// Robot Parameter                         
UserData.DelayTime                         := _parCfg.Rob.Parameter.DelayTime;
UserData.WaitForNrOfCmd                    := _parCfg.Rob.Parameter.WaitForNrOfCmd;
UserData.WaitAtBlendingZone                := _parCfg.Rob.Parameter.WaitAtBlendingZone;
UserData.AllowSecSeqWhileSubprogram        := _parCfg.Rob.Parameter.AllowSecSeqWhileSubprogram;
UserData.AllowDynamicBlending              := _parCfg.Rob.Parameter.AllowDynamicBlending;
UserData.SyncReaction                      := _parCfg.Rob.Parameter.SyncReaction;
UserData.SyncDelay                         := _parCfg.Rob.Parameter.SyncDelay;
UserData.MessageLevel                      := _parcfg.Rob.Parameter.MessageLevel;

// ReadRobotData
UserData.RCManufacturer                    := AxesGroup.State.RobotData.RCManufacturer; 
UserData.RCOrderID                         := AxesGroup.State.RobotData.RCOrderID; 
UserData.RCSerialNumber                    := AxesGroup.State.RobotData.RCSerialNumber;
UserData.RASerialNumber                    := AxesGroup.State.RobotData.RASerialNumber;
UserData.RCFirmwareVersion                 := AxesGroup.State.RobotData.RCFirmwareVersion;

UserData.RCInterpreterVersion.MajorVersion := STRING_TO_USINT(MID(AxesGroup.State.RobotData.RCInterpreterVersion, LEN := 1, POS := 1));
UserData.RCInterpreterVersion.MinorVersion := STRING_TO_USINT(MID(AxesGroup.State.RobotData.RCInterpreterVersion, LEN := 1, POS := 2));
UserData.RCInterpreterVersion.PatchVersion := STRING_TO_USINT(MID(AxesGroup.State.RobotData.RCInterpreterVersion, LEN := 1, POS := 3));

UserData.AxisJointUsed                     := AxesGroup.State.RobotData.AxisJointUsed;
UserData.AxisExternalUsed                  := AxesGroup.State.RobotData.AxisExternalUsed;
UserData.AxisJointUnit                     := AxesGroup.State.RobotData.AxisJointUnit;
UserData.AxisExternalUnit                  := AxesGroup.State.RobotData.AxisExternalUnit;
UserData.RCSupportedFunctions              := AxesGroup.State.RobotData.RCSupportedFunctions;
                                           
UserData.BrakeTestRequired                 := AxesGroup.State.ConfigurationData.BrakeTestRequired;
UserData.PathAccuracyMode                  := AxesGroup.State.ConfigurationData.PathAccuracyMode;
UserData.AvoidSingularity                  := AxesGroup.State.ConfigurationData.AvoidSingularity;
UserData.ConstantVelocitySupported         := AxesGroup.State.ConfigurationData.ConstantVelocitySupported;
UserData.StepModeExactStopActive           := AxesGroup.State.ConfigurationData.StepModeExactStopActive;
UserData.StepModeBlendingActive            := AxesGroup.State.ConfigurationData.StepModeBlendingActive;
UserData.AcceleratingSupported             := AxesGroup.State.ConfigurationData.AcceleratingSupported;
UserData.DeceleratingSupported             := AxesGroup.State.ConfigurationData.DecceleratingSupported;
                                           
UserData.Initialized                       := Initialized;
UserData.Synchronized                      := Synchronized;
                                           
// Cyclic data                             
UserData.RCSRCIVersion                     := AxesGroup.Cyclic.RobToPlc.SRCIVersion;
UserData.IsMoving                          := AxesGroup.Cyclic.RobToPlc.StatusRobotArm.IsMoving;
UserData.PrimarySequencePaused             := AxesGroup.Cyclic.RobToPlc.StatusRobotArm.PrimarySequencePaused;
UserData.InPrimaryPos                      := AxesGroup.Cyclic.RobToPlc.StatusRobotArm.InPrimaryPos;
UserData.SecondarySequenceActive           := AxesGroup.Cyclic.RobToPlc.StatusRobotArm.SecondarySequenceActive;
UserData.ErrorPending                      := AxesGroup.Cyclic.RobToPlc.StatusRobotArm.ErrorPending;
UserData.RestartInProgress                 := AxesGroup.Cyclic.RobToPlc.StatusRobotArm.RestartInProgress;
UserData.Enabled                           := AxesGroup.Cyclic.RobToPlc.StatusRobotArm.Enabled;
UserData.Idle                              := AxesGroup.Cyclic.RobToPlc.StatusRobotArm.RaSequenceState = RaSequenceState.IDLE;
UserData.Executing                         := AxesGroup.Cyclic.RobToPlc.StatusRobotArm.RaSequenceState = RaSequenceState.EXECUTING;
UserData.Interrupted                       := AxesGroup.Cyclic.RobToPlc.StatusRobotArm.RaSequenceState = RaSequenceState.INTERRUPTED;
UserData.IsBlending                        := AxesGroup.Cyclic.RobToPlc.StatusRobotArm.IsBlending;  
UserData.OperationMode                     := AxesGroup.Cyclic.RobToPlc.StatusRobotArm.OperationMode;
UserData.CollisionDetectionEnabled         := AxesGroup.Cyclic.RobToPlc.StatusRobotArm.CollisionDetectedEnabled;
UserData.CollisionDetected                 := AxesGroup.Cyclic.RobToPlc.StatusRobotArm.CollisionDetected;
UserData.RestartRequested                  := AxesGroup.Cyclic.RobToPlc.StatusRobotArm.RestartRequested;
UserData.Accelerating                      := AxesGroup.Cyclic.RobToPlc.StatusRobotArm.Accelerating;
UserData.Decelerating                      := AxesGroup.Cyclic.RobToPlc.StatusRobotArm.Decelerating;
UserData.ConstantVelocity                  := AxesGroup.Cyclic.RobToPlc.StatusRobotArm.ConstantVelocity;
UserData.ActualOverride                    := PERCENT_UINT_TO_REAL( Value := AxesGroup.Cyclic.RobToPlc.Override, IsOptional := FALSE);

// Cyclic optional data
UserData.CartesianPosition                 := AxesGroup.CyclicOptional.RobToPlc.CartesianPosition;
UserData.ExtCartesianPosition              := AxesGroup.CyclicOptional.RobToPlc.CartesianPositionExt;  
UserData.JointPosition                     := AxesGroup.CyclicOptional.RobToPlc.JointPosition;
UserData.ExtJointPosition                  := AxesGroup.CyclicOptional.RobToPlc.JointPositionExt;

// Synchronizing
UserData.ToolDataSynchronizing             := AxesGroup.State.Synchronizing.Tool;
UserData.FrameDataSynchronizing            := AxesGroup.State.Synchronizing.Frame;
UserData.LoadDataSynchronizing             := AxesGroup.State.Synchronizing.Load;
UserData.WorkAreaDataSynchronizing         := AxesGroup.State.Synchronizing.WorkAreas;
UserData.SWLimitsSynchronizing             := AxesGroup.State.Synchronizing.SwLimits;
UserData.DefaultDynamicsSynchronizing      := AxesGroup.State.Synchronizing.DefaultDynamics;
UserData.ReferenceDynamicsSynchronizing    := AxesGroup.State.Synchronizing.ReferenceDynamics;


UserData.ActivateTwoSequences              := _parCfg.Com.TwoSequences;
UserData.ReadingCartesianPosition          :=  AxesGroup.State.ReadingCartesianPosition;
UserData.ReadingExtCartesianPosition       :=  AxesGroup.State.ReadingCartesianPositionExt;
UserData.ReadingJointPosition              :=  AxesGroup.State.ReadingJointPosition;
UserData.ReadingExtJointPosition           :=  AxesGroup.State.ReadingJointPositionExt;

                
END_METHOD

METHOD PRIVATE OnCall
VAR_IN_OUT
   /// Robot assignment of function
  AxesGroup : AxesGroup;
END_VAR
                  // map numeric value to enum, so that the corresponding message text is directly shown by the tooltip
ErrorIdEnum   := ErrorId;
WarningIdEnum := WarningId;
InfoIdEnum    := InfoId;

Error := HasError;

// Check Payload and In/Out data size
IF (( ROBOT_IN_DATA_SIZE  < 64 ) OR
    ( ROBOT_OUT_DATA_SIZE < 64 ))
THEN
  SetError(ErrorID := RobotLibraryErrorIdEnum.ERR_INVALID_LIBRARY_PARA, Overwrite := TRUE );
  RETURN;
END_IF


// Check AxesGroupID valid
IF (( AxesGroupID < RobotLibraryConstants.AXES_GROUP_ID_MIN ) OR
    ( AxesGroupID > RobotLibraryConstants.AXES_GROUP_ID_MAX ))
THEN
  SetError( ErrorID := RobotLibraryErrorIdEnum.ERR_INVALID_AXES_GROUP_ID, Overwrite := TRUE );
  RETURN;
END_IF


// Reset flag for initialization / Synchronization
IF ( Initialized OR Synchronized) AND ( AxesGroup.Cyclic.RobToPlc.TelegramState <> TelegramState.INITIALIZED)
THEN
  // Reset initialized flag
  Initialized := FALSE;
  // Reset Synchronized flag
  Synchronized := FALSE;
  // Set error 
  SetError( ErrorID := RobotLibraryErrorIdEnum.ERR_INIT_LOST_UNKNOWN_0x80A2, Overwrite := TRUE );
END_IF


// Warning for ACR Registers running low
IF ( AxesGroup.Acyclic.ActiveCommandRegister.CurrentAcrUsagePercent > RobotLibraryParameter.ACR_USAGE_WARNING_LIMIT )
THEN
  SetWarning( WarningID := RobotLibraryWarningIdEnum.WARN_ACR_FREE_ENTRIES_LOW, Overwrite := TRUE);  
END_IF

// Check ToolData boundary
IF ( AxesGroup.SystemData.ToolDataMin  <> 0 )  
THEN
  SetWarning( WarningID := RobotLibraryWarningIdEnum.WARN_TOOL_DATA_ARRAY_NOT_START_AT_ZERO, Overwrite := FALSE );
END_IF

// Check FrameData boundary
IF ( AxesGroup.SystemData.FrameDataMin <> 0 ) AND ( NOT HasWarning )  
THEN
  SetWarning( WarningID := RobotLibraryWarningIdEnum.WARN_FRAME_DATA_ARRAY_NOT_START_AT_ZERO, Overwrite := FALSE );
END_IF

// Check WorkAreas boundary
IF ( AxesGroup.SystemData.WorkAreasMin <> 0 ) AND ( NOT HasWarning )  
THEN
  SetWarning( WarningID := RobotLibraryWarningIdEnum.WARN_FRAME_DATA_ARRAY_NOT_START_AT_ZERO, Overwrite := FALSE);
END_IF


// Check configuration parameter changed ? 
CheckParameterChanged(AxesGroup := AxesGroup);
                
END_METHOD

METHOD OnExecRun : DINT
VAR_IN_OUT
  /// Robot assignment of function
  AxesGroup         : AxesGroup;
END_VAR
                  // building rising and falling edges
_enable_R( CLK := Enable);
_enable_F( CLK := Enable);

IF ( _enable_F.Q)
THEN
  Reset(AxesGroup := AxesGroup);
END_IF


OnExecRun := RobotLibraryConstants.RUNNING;

CASE _stepCmd OF
  
  00:  IF ( _enable_R.Q )
       THEN
         // Create log entry
         CreateLogMessage ( Timestamp   := SystemTime,
                            MessageType := MessageType.CMD,
                            Severity    := Severity.INFO,
                            MessageCode := 0,
                            MessageText := 'Robot Task Enabled');
       
         // reset the rising edge
        _enable_R();
         // set busy flag
         Busy := TRUE;
         // set timeout
         SetTimeout(PT := _timeoutCmd, rTimer := _timerCmd);
         // Reset FastStop       
         AxesGroup.Cyclic.PlcToRob.FastStop := 0;
         // Reset Active command register
         AxesGroup.Acyclic.ActiveCommandRegister.Reset();
       
         // check parameter valid
         IF ( CheckParameterValid(AxesGroup := AxesGroup) )
         THEN
           // take configuration parameter if not yet enabled
          _parCfg := ParCfg;
           // inc step counter
          _stepCmd := _stepCmd + 1; 
         END_IF
       END_IF
     
  01:  CASE AxesGroup.Cyclic.RobToPlc.TelegramState  OF

         TelegramState.UNDEFINED : ;
         
         TelegramState.ERROR_161_TELEGRAM_CONTROL_MISMATCH_TELEGRAM_STATE..TelegramState.ERROR_172_TELEGRAM_NUMBER_NOT_SUPPORTED:

           // clear error
           AxesGroup.Cyclic.PlcToRob.Control := ControlHalfByte.ACK_ERROR;        
           AxesGroup.Cyclic.PlcToRob.Control := ControlHalfByte.RESET; // always a reset, so that on the robot side the ACR is reseted         

         TelegramState.ERROR_173_SERVER_CONNECTION_LOST:

           // Reset interface including the ACR register on server side
           AxesGroup.Cyclic.PlcToRob.Control := ControlHalfByte.RESET;        
           
         TelegramState.READY_TO_RESUME :  
         
           // Resume
           AxesGroup.Cyclic.PlcToRob.Control := ControlHalfByte.RESUME;        
         
         TelegramState.READY_FOR_INITIALIZATION: 

           // Request initialization
           AxesGroup.Cyclic.PlcToRob.Control := ControlHalfByte.INITIALIZE;
           
         TelegramState.INITIALIZED: 

           // Reset Telegram Control 
           AxesGroup.Cyclic.PlcToRob.Control := ControlHalfByte.NONE;
           
           // Check SRCI Version is compatible ? 
           IF ( AxesGroup.Cyclic.RobToPlc.SRCIVersion.MajorVersion = RobotLibraryConstants.SRCIVersion.MajorVersion )
           THEN
             // set timeout
             SetTimeout(PT := _timeoutCmd, rTimer := _timerCmd);
             // inc step counter
            _stepCmd := _stepCmd + 1; 
           ELSE
             // set error 
             ErrorID     := RobotLibraryErrorIdEnum.ERR_SRCI_MAJOR_VERSION_INCOMPATIBLE_0x80A4;
             ErrorAddTxt := CONCAT('_stepCmd = ' , DINT_TO_STRING(_stepCmd));
           END_IF

       ELSE
         // TelegrammState in error          
         SetError( ErrorID := RobotLibraryErrorIdEnum.ERR_INIT_LOST_UNKNOWN_0xA2, Overwrite := TRUE );
         ErrorAddTxt := CONCAT('_stepCmd = ' , DINT_TO_STRING(_stepCmd));
       END_CASE

       // timeout exceeded ? 
       IF (CheckTimeout(_timerCmd) = RobotLibraryConstants.OK)
       THEN
         // Check Telegram State error ? 
         IF (( AxesGroup.Cyclic.RobToPlc.TelegramState >= TelegramState.ERROR_161_TELEGRAM_CONTROL_MISMATCH_TELEGRAM_STATE ) OR
             ( AxesGroup.Cyclic.RobToPlc.TelegramState <= TelegramState.ERROR_173_SERVER_CONNECTION_LOST                   ))
         THEN
           ErrorID     := AxesGroup.Cyclic.RobToPlc.TelegramState;
           ErrorAddTxt := CONCAT('_stepCmd = ' , DINT_TO_STRING(_stepCmd));
         ELSE
           ErrorID     := RobotLibraryErrorIdEnum.ERR_TIMEOUT_CMD;
           ErrorAddTxt := CONCAT('_stepCmd = ' , DINT_TO_STRING(_stepCmd));
         END_IF
       END_IF

       
  02: IF (( NOT _readMessages.Busy  ) AND 
          ( NOT _readMessages.Error )) 
      THEN
        // start function block
       _readMessages.Enable := TRUE;
       _readMessages.ParCmd.MsgID := 0;
       _readMessages.ParCmd.MessageLevel := _parCfg.Rob.Parameter.MessageLevel;
        
        // set timeout
        SetTimeout(PT := _timeoutCmd, rTimer := _timerCmd);
        // inc step counter
       _stepCmd := _stepCmd + 1;       
      ELSE
        // check error ? 
        IF (_readMessages.Error)
        THEN
          ErrorID     := _readMessages.ErrorID;
          ErrorAddTxt := _readMessages.ErrorAddTxt;;
        END_IF  
        // timeout exceeded ? 
        IF (CheckTimeout(_timerCmd) = RobotLibraryConstants.OK)
        THEN
          ErrorID     := RobotLibraryErrorIdEnum.ERR_TIMEOUT_CMD;
          ErrorAddTxt := CONCAT('_stepCmd = ' , DINT_TO_STRING(_stepCmd));
        END_IF
      END_IF
  
  03: IF ((     _readMessages.Enabled ) AND
          ( NOT _readMessages.Error   ))
      THEN       
        // --------------------------------------------------------------- 
        // !!! ReadMessages must stay active for the Message mechanism !!!
        // --------------------------------------------------------------- 
        // ReadMessages.Enable := FALSE;  
        // set timeout
        SetTimeout(PT := _timeoutCmd, rTimer := _timerCmd);
        // inc step counter
       _stepCmd := _stepCmd + 1;
      ELSE
         // check error ? 
         IF (_readMessages.Error)
         THEN
           ErrorID     := _readMessages.ErrorID;
           ErrorAddTxt := _readMessages.ErrorAddTxt;;
         END_IF  
       
         // timeout exceeded ? 
         IF (CheckTimeout(_timerCmd) = RobotLibraryConstants.OK)
         THEN
           ErrorID     := RobotLibraryErrorIdEnum.ERR_TIMEOUT_CMD;
           ErrorAddTxt := CONCAT('_stepCmd = ' , DINT_TO_STRING(_stepCmd));
         END_IF
       END_IF       
       
       
  04: IF (( NOT _exchangeConfiguration.Busy  ) AND 
          ( NOT _exchangeConfiguration.Error ))
      THEN
        // set command parameter
       _exchangeConfiguration.ParCmd.LogLevel                           :=  LogLevel; 
       _exchangeConfiguration.ParCmd.WaitAtBlendingZone                 := _parCfg.Rob.Parameter.WaitAtBlendingZone;
       _exchangeConfiguration.ParCmd.AllowSecSeqWhileSubprogram         := _parCfg.Rob.Parameter.AllowSecSeqWhileSubprogram;
       _exchangeConfiguration.ParCmd.AllowDynamicBlending               := _parCfg.Rob.Parameter.AllowDynamicBlending;
       _exchangeConfiguration.ParCmd.DelayTime                          := _parCfg.Rob.Parameter.DelayTime;
       _exchangeConfiguration.ParCmd.WaitForNrOfCmd                     := _parCfg.Rob.Parameter.WaitForNrOfCmd;
       _exchangeConfiguration.ParCmd.LifeSignTimeOut                    :=  TIME_TO_UINT(_parCfg.Com.LifeSignTimeOut);
       _exchangeConfiguration.ParCmd.SyncDelay                          := _parCfg.Rob.Parameter.SyncDelay;
       _exchangeConfiguration.ParCmd.SyncReaction                       := _parCfg.Rob.Parameter.SyncReaction;
       _exchangeConfiguration.ParCmd.DataEnableSync                     :=  SyncModesToDataEnableSync(Value := _parCfg.Plc.Parameter.SynchronizationModes);
       _exchangeConfiguration.ParCmd.DataInSync.ToolsInSync             :=  FALSE;
       _exchangeConfiguration.ParCmd.DataInSync.FramesInSync            :=  FALSE;
       _exchangeConfiguration.ParCmd.DataInSync.LoadsInSync             :=  FALSE;
       _exchangeConfiguration.ParCmd.DataInSync.WorkAreasInSync         :=  FALSE;
       _exchangeConfiguration.ParCmd.DataInSync.SoftwareLimitsInSync    :=  FALSE;
       _exchangeConfiguration.ParCmd.DataInSync.DefaultDynamicsInSync   :=  FALSE;
       _exchangeConfiguration.ParCmd.DataInSync.ReferenceDynamicsInSync :=  FALSE;         
       
        // start function block
       _exchangeConfiguration.Enable := TRUE;
        // set timeout
        SetTimeout(PT := _timeoutCmd, rTimer := _timerCmd);
        // inc step counter
       _stepCmd := _stepCmd + 1;       
      ELSE
        // check error ? 
        IF (_exchangeConfiguration.Error)
        THEN
          ErrorID     := _exchangeConfiguration.ErrorID;
          ErrorAddTxt := _exchangeConfiguration.ErrorAddTxt;;
        END_IF  
       
        // timeout exceeded ? 
        IF (CheckTimeout(_timerCmd) = RobotLibraryConstants.OK)
        THEN
          ErrorID     := RobotLibraryErrorIdEnum.ERR_TIMEOUT_CMD;
          ErrorAddTxt := CONCAT('_stepCmd = ' , DINT_TO_STRING(_stepCmd));
        END_IF
      END_IF
  
  
  05: IF ((     _exchangeConfiguration.Enabled ) AND
          ( NOT _exchangeConfiguration.Error   ))
      THEN     
        // --------------------------------------------------------------------- 
        // !!! ExchangeConfiguration must stay active for the Sync mechanism !!!
        // --------------------------------------------------------------------- 
        // ExchangeConfiguration.Enable := FALSE;  
        // set timeout
        SetTimeout(PT := _timeoutCmd, rTimer := _timerCmd);
        // inc step counter
       _stepCmd := _stepCmd + 1;       
      ELSE
        // check error ? 
        IF (_exchangeConfiguration.Error)
        THEN
          ErrorID     := _exchangeConfiguration.ErrorID;
          ErrorAddTxt := _exchangeConfiguration.ErrorAddTxt;;
        END_IF  
       
        // timeout exceeded ? 
        IF (CheckTimeout(_timerCmd) = RobotLibraryConstants.OK)
        THEN
          ErrorID     := RobotLibraryErrorIdEnum.ERR_TIMEOUT_CMD;
          ErrorAddTxt := CONCAT('_stepCmd = ' , DINT_TO_STRING(_stepCmd));
        END_IF
      END_IF

       
  06: IF (( NOT _readRobotData.Busy  ) AND 
          ( NOT _readRobotData.Error )) 
      THEN
        // start function block
       _readRobotData.Execute := TRUE;
        // set timeout
        SetTimeout(PT := _timeoutCmd, rTimer := _timerCmd);
        // inc step counter
       _stepCmd := _stepCmd + 1;       
      ELSE
        // check error ? 
        IF (_readRobotData.Error)
        THEN
          ErrorID     := _readRobotData.ErrorID;
          ErrorAddTxt := _readRobotData.ErrorAddTxt;;
        END_IF  
        // timeout exceeded ? 
        IF (CheckTimeout(_timerCmd) = RobotLibraryConstants.OK)
        THEN
          ErrorID     := RobotLibraryErrorIdEnum.ERR_TIMEOUT_CMD;
          ErrorAddTxt := CONCAT('_stepCmd = ' , DINT_TO_STRING(_stepCmd));
        END_IF
      END_IF
    
  
  07: IF ((     _readRobotData.Done  ) AND
          ( NOT _readRobotData.Busy  ) AND
          ( NOT _readRobotData.Error ))          
      THEN       
        // set initialized flag
        Initialized := TRUE;       
        // start function block
       _readRobotData.Execute := FALSE;
        // set timeout
        SetTimeout(PT := _timeoutCmd, rTimer := _timerCmd);
        // inc step counter
       _stepCmd := _stepCmd + 1;
       ELSE
         // check error ? 
         IF (_readRobotData.Error)
         THEN
           ErrorID     := _readRobotData.ErrorID;
           ErrorAddTxt := _readRobotData.ErrorAddTxt;;
         END_IF  
       
         // timeout exceeded ? 
         IF (CheckTimeout(_timerCmd) = RobotLibraryConstants.OK)
         THEN
           ErrorID     := RobotLibraryErrorIdEnum.ERR_TIMEOUT_CMD;
           ErrorAddTxt := CONCAT('_stepCmd = ' , DINT_TO_STRING(_stepCmd));
         END_IF
       END_IF

       
  08:  // Update Initialized state
       Initialized := NOT ERROR AND NOT Synchronized; {warning 'ToDo'}
       Initialized := NOT Synchronized;

       // Wait for task disable
       IF ( NOT Enable)
       THEN
         // Reset active command register
         AxesGroup.Acyclic.ActiveCommandRegister.Reset();
         // reset internal variables
         Reset(AxesGroup := AxesGroup);
         // Reset step counter
        _stepCmd := 0;         
         // finished okay
         OnExecRun := RobotLibraryConstants.OK;
       END_IF  

       
ELSE
  // invalid step
  ErrorID     := RobotLibraryErrorIdEnum.ERR_INVALID_STEP;
  ErrorAddTxt := CONCAT('_stepCmd = ' , DINT_TO_STRING(_stepCmd));
END_CASE
                
END_METHOD

METHOD PRIVATE ParseRecvPayload
VAR_IN_OUT
  /// Robot assignment of function
  AxesGroup   : AxesGroup;
  /// Inputs of PLC for communication from RC
  RobotInData : ARRAY[*] OF BYTE;
END_VAR
                  // reset all variables and payload
RecvData.Reset();
// Call RecvData FB, update payload and size 
RecvData(Payload := RobotInData, PayloadSize := ROBOT_IN_DATA_SIZE);

// check new data to receive ? 
IF ( Telegram.RobToPlc.Sequence[0].Header.SEQ_ACK <> AxesGroup.State.LastACK[0]) {warning 'ToDo: handle 2nd sequence'} 
THEN
  // delete old telegram data 
  SysDepMemSet(pDest := ADR(Telegram.RobToPlc), Value := 0 , DataLen := SIZEOF(Telegram.RobToPlc));
END_IF


ParseRecvPayloadHeader        ( AxesGroup := AxesGroup);
ParseRecvPayloadCyclic        ( AxesGroup := AxesGroup);
ParseRecvPayloadCyclicOptional( AxesGroup := AxesGroup);
ParseRecvPayloadSequence      ( AxesGroup := AxesGroup);
ParseRecvPayloadFooter        ( AxesGroup := AxesGroup);
ParseRecvPayloadLogging       ( AxesGroup := AxesGroup);


AxesGroup.State.LastACK[0] := Telegram.RobToPlc.Sequence[0].Header.SEQ_ACK; 
AxesGroup.State.LastACK[1] := Telegram.RobToPlc.Sequence[1].Header.SEQ_ACK; 
                
END_METHOD

METHOD PRIVATE ParseRecvPayloadCyclic
VAR_IN_OUT
  /// Robot assignment of function
  AxesGroup: AxesGroup;
END_VAR
                  
                
END_METHOD

METHOD PRIVATE ParseRecvPayloadCyclicOptional
VAR_IN_OUT
  /// Robot assignment of function
  AxesGroup    : AxesGroup;
END_VAR

VAR 
  /// internal index for loops
 _idx : DINT;
END_VAR
                  // AxesGroup.OptionalCyclic.RobToPlc.SubProgramData {{{
IF ( AxesGroup.CyclicOptional.RobToPlc.SubProgramData.Active )
THEN
  FOR _idx := 0 TO 25 {warning 'Add contant for DataMax'}
  DO
    Telegram.RobToPlc.CyclicOptional.SubProgramData.Data[_idx] := RecvData.GetByte(); 
  END_FOR
END_IF
// }}}
  
// AxesGroup.OptionalCyclic.RobToPlc.CartesianPos {{{
IF ( AxesGroup.CyclicOptional.RobToPlc.CartesianPosition.Active )
THEN
  Telegram.RobToPlc.CyclicOptional.CartesianPosition.X                    := RecvData.GetReal();
  Telegram.RobToPlc.CyclicOptional.CartesianPosition.Y                    := RecvData.GetReal();
  Telegram.RobToPlc.CyclicOptional.CartesianPosition.Z                    := RecvData.GetReal();
  Telegram.RobToPlc.CyclicOptional.CartesianPosition.Rx                   := RecvData.GetReal();
  Telegram.RobToPlc.CyclicOptional.CartesianPosition.Ry                   := RecvData.GetReal();
  Telegram.RobToPlc.CyclicOptional.CartesianPosition.Rz                   := RecvData.GetReal();
  Telegram.RobToPlc.CyclicOptional.CartesianPosition.Config               := RecvData.GetWord();
  Telegram.RobToPlc.CyclicOptional.CartesianPosition.Turns_J2_J1          := RecvData.GetByte();
  Telegram.RobToPlc.CyclicOptional.CartesianPosition.Turns_J4_J3          := RecvData.GetByte();
  Telegram.RobToPlc.CyclicOptional.CartesianPosition.Turns_J6_J5          := RecvData.GetByte();
  Telegram.RobToPlc.CyclicOptional.CartesianPosition.Turns_E1             := RecvData.GetByte();  
  Telegram.RobToPlc.CyclicOptional.CartesianPosition.E1                   := RecvData.GetReal();  
  Telegram.RobToPlc.CyclicOptional.CartesianPosition.ToolNo               := RecvData.GetUsint();
  Telegram.RobToPlc.CyclicOptional.CartesianPosition.FrameNo              := RecvData.GetUsint();
  Telegram.RobToPlc.CyclicOptional.CartesianPosition.CurrentlyUsedToolNo  := RecvData.GetUsint();
  Telegram.RobToPlc.CyclicOptional.CartesianPosition.CurrentlyUsedFrameNo := RecvData.GetUsint();
  Telegram.RobToPlc.CyclicOptional.CartesianPosition.Reserve_1            := RecvData.GetByte();
  Telegram.RobToPlc.CyclicOptional.CartesianPosition.Reserve_2            := RecvData.GetByte();  
END_IF
// }}}

// AxesGroup.OptionalCyclic.RobToPlc.JointPosition {{{
IF ( AxesGroup.CyclicOptional.RobToPlc.JointPosition.Active )
THEN
  Telegram.RobToPlc.CyclicOptional.JointPosition.J1         := RecvData.GetReal();
  Telegram.RobToPlc.CyclicOptional.JointPosition.J2         := RecvData.GetReal();
  Telegram.RobToPlc.CyclicOptional.JointPosition.J3         := RecvData.GetReal();
  Telegram.RobToPlc.CyclicOptional.JointPosition.J4         := RecvData.GetReal();
  Telegram.RobToPlc.CyclicOptional.JointPosition.J5         := RecvData.GetReal();
  Telegram.RobToPlc.CyclicOptional.JointPosition.J6         := RecvData.GetReal();
  Telegram.RobToPlc.CyclicOptional.JointPosition.E1         := RecvData.GetReal();
  Telegram.RobToPlc.CyclicOptional.JointPosition.E1_Reserve := RecvData.GetWord();
END_IF  
// }}}

// AxesGroup.OptionalCyclic.RobToPlc.CartesianForce {{{
IF ( AxesGroup.CyclicOptional.RobToPlc.Force.Active )
THEN
  Telegram.RobToPlc.CyclicOptional.Force.X  := RecvData.GetReal();
  Telegram.RobToPlc.CyclicOptional.Force.Y  := RecvData.GetReal();
  Telegram.RobToPlc.CyclicOptional.Force.Z  := RecvData.GetReal();
  Telegram.RobToPlc.CyclicOptional.Force.Rx := RecvData.GetReal();
  Telegram.RobToPlc.CyclicOptional.Force.Ry := RecvData.GetReal();
  Telegram.RobToPlc.CyclicOptional.Force.Rz := RecvData.GetReal();
END_IF  
// }}}    
  
// AxesGroup.OptionalCyclic.RobToPlc.Current {{{
IF ( AxesGroup.CyclicOptional.RobToPlc.Current.Active )
THEN
  Telegram.RobToPlc.CyclicOptional.Current.J1  := RecvData.GetReal();
  Telegram.RobToPlc.CyclicOptional.Current.J2  := RecvData.GetReal();
  Telegram.RobToPlc.CyclicOptional.Current.J3  := RecvData.GetReal();
  Telegram.RobToPlc.CyclicOptional.Current.J4  := RecvData.GetReal();
  Telegram.RobToPlc.CyclicOptional.Current.J5  := RecvData.GetReal();
  Telegram.RobToPlc.CyclicOptional.Current.J6  := RecvData.GetReal();
END_IF    
  
// AxesGroup.OptionalCyclic.RobToPlc.CartesianPosExt {{{
IF ( AxesGroup.CyclicOptional.RobToPlc.CartesianPositionExt.Active )
THEN
  Telegram.RobToPlc.CyclicOptional.CartesianPositionExt.E2 := RecvData.GetReal();
  Telegram.RobToPlc.CyclicOptional.CartesianPositionExt.E3 := RecvData.GetReal();
  Telegram.RobToPlc.CyclicOptional.CartesianPositionExt.E4 := RecvData.GetReal();
  Telegram.RobToPlc.CyclicOptional.CartesianPositionExt.E5 := RecvData.GetReal();
  Telegram.RobToPlc.CyclicOptional.CartesianPositionExt.E6 := RecvData.GetReal();
END_IF  
// }}}       
  
// AxesGroup.OptionalCyclic.RobToPlc.JointPosition {{{
IF ( AxesGroup.CyclicOptional.RobToPlc.JointPositionExt.Active )
THEN
  Telegram.RobToPlc.CyclicOptional.JointPositionExt.E2 := RecvData.GetReal();
  Telegram.RobToPlc.CyclicOptional.JointPositionExt.E3 := RecvData.GetReal();
  Telegram.RobToPlc.CyclicOptional.JointPositionExt.E4 := RecvData.GetReal();
  Telegram.RobToPlc.CyclicOptional.JointPositionExt.E5 := RecvData.GetReal();
  Telegram.RobToPlc.CyclicOptional.JointPositionExt.E6 := RecvData.GetReal();  
END_IF  
// }}}    
      
// AxesGroup.OptionalCyclic.RobToPlc.CartesianForceExt {{{
IF ( AxesGroup.CyclicOptional.RobToPlc.ForceExt.Active )
THEN
  Telegram.RobToPlc.CyclicOptional.ForceExt.E1  := RecvData.GetReal();
  Telegram.RobToPlc.CyclicOptional.ForceExt.E2  := RecvData.GetReal();
  Telegram.RobToPlc.CyclicOptional.ForceExt.E3  := RecvData.GetReal();
  Telegram.RobToPlc.CyclicOptional.ForceExt.E4  := RecvData.GetReal();
  Telegram.RobToPlc.CyclicOptional.ForceExt.E5  := RecvData.GetReal();
  Telegram.RobToPlc.CyclicOptional.ForceExt.E6  := RecvData.GetReal();
END_IF
// }}}    
  
// AxesGroup.OptionalCyclic.RobToPlc.CurrentExt {{{
IF ( AxesGroup.CyclicOptional.RobToPlc.CurrentExt.Active )
THEN
  Telegram.RobToPlc.CyclicOptional.CurrentExt.E1  := RecvData.GetReal();
  Telegram.RobToPlc.CyclicOptional.CurrentExt.E2  := RecvData.GetReal();
  Telegram.RobToPlc.CyclicOptional.CurrentExt.E3  := RecvData.GetReal();
  Telegram.RobToPlc.CyclicOptional.CurrentExt.E4  := RecvData.GetReal();
  Telegram.RobToPlc.CyclicOptional.CurrentExt.E5  := RecvData.GetReal();
  Telegram.RobToPlc.CyclicOptional.CurrentExt.E6  := RecvData.GetReal();
END_IF
// }}}
                
END_METHOD

METHOD PRIVATE ParseRecvPayloadFooter
VAR_IN_OUT
  /// Robot assignment of function
  AxesGroup : AxesGroup;
END_VAR
                  Telegram.RobToPlc.Footer.LifeSign := RecvData.GetLifeSignFooter(); 

                
END_METHOD

METHOD PRIVATE ParseRecvPayloadHeader
VAR_IN_OUT
  /// Robot assignment of function
  AxesGroup    : AxesGroup;
END_VAR
                  // Version
Telegram.RobToPlc.Header.SRCIVersion := ByteToVersion(RecvData.GetByte());
// Connection alive signal
Telegram.RobToPlc.Header.LifeSign    := RecvData.GetHalfeByte2(IncPayloadPtr := TRUE);
// Reserved byte
Telegram.RobToPlc.Header.Reserved       := RecvData.GetByte();
// Initialization and Telegram control state
Telegram.RobToPlc.Header.TelegramState  := RecvData.GetUsint();
// Combination of various RA related states.
Telegram.RobToPlc.Header.StatusRobotArm := RecvData.GetDword();
// Actual override in percentage encoding 
Telegram.RobToPlc.Header.Override       := RecvData.GetUint();
                
END_METHOD

METHOD PRIVATE ParseRecvPayloadLogging
VAR_IN_OUT
  /// Robot assignment of function
  AxesGroup    : AxesGroup;
END_VAR

VAR
  /// internal sequence index for loops
  _seqIdx : DINT;
  /// internal fragment index for loops
  _fragIdx : DINT;
END_VAR
                  RETURN;
FOR _seqIdx := 0 TO AxesGroup.State.SequenceCountRecv
DO
  // check new data to receive ? 
  IF ( Telegram.RobToPlc.Sequence[_seqIdx].Header.SEQ_ACK <> AxesGroup.State.LastACK[_seqIdx]) 
  THEN
    // Check sequence payload > 0 ?    
    IF (Telegram.RobToPlc.Sequence[_seqIdx].Header.PayloadLength > 0)
    THEN
      // Create log entry
      CreateLogMessagePara4 ( Timestamp   := SystemTime,
                              MessageType := MessageType.CMD,
                              Severity    := Severity.DEBUG,
                              MessageCode := 0,
                              MessageText := 'RecvData: ACK = {1}, received Sequence [{2}] with PayloadLength = {3}, Lifesign = {4}',
                              Para1       :=  UINT_TO_STRING(Telegram.RobToPlc.Sequence[_seqIdx].Header.SEQ_ACK),
                              Para2       :=  DINT_TO_STRING(_seqIdx),
                              Para3       :=  UINT_TO_STRING(Telegram.RobToPlc.Sequence[_seqIdx].Header.PayloadLength),
                              Para4       :=  BYTE_TO_STRING(Telegram.RobToPlc.Header.LifeSign));
  
      FOR _fragIdx := 0 TO AxesGroup.State.FragmentCountRecv[_seqIdx] 
      DO
        // Check fragment payload > 0 ?    
        IF (Telegram.RobToPlc.Sequence[_seqIdx].Fragment[_fragIdx].Header.PayloadLength > 0)
        THEN
          // Create log entry
          CreateLogMessagePara5 ( Timestamp   := SystemTime,
                                  MessageType := MessageType.CMD,
                                  Severity    := Severity.DEBUG,
                                  MessageCode := 0,
                                  MessageText := 'RecvData: received Fragment [{1}] with PayloadLength = {2}, CmdID <{3}> , CmdState: {4}, Fragment-Action Bits: {5}',
                                  Para1       :=  DINT_TO_STRING(0), {warning 'Add seqIdx'}
                                  Para2       :=  UINT_TO_STRING              (Telegram.RobToPlc.Sequence[_seqIdx].Fragment[_fragIdx].Header.PayloadLength),
                                  Para3       :=  DINT_TO_STRING              (Telegram.RobToPlc.Sequence[_seqIdx].Fragment[_fragIdx].Header.CmdID),
                                  Para4       :=  CMD_MESSAGE_STATE_TO_STRING (Telegram.RobToPlc.Sequence[_seqIdx].Fragment[_fragIdx].Command.Header.State),
                                  Para5       :=    FRAGMENT_ACTION_TO_STRING (Telegram.RobToPlc.Sequence[_seqIdx].Fragment[_fragIdx].Header.FragmentAction));
        END_IF
      END_FOR    
    END_IF
  END_IF
END_FOR  
                
END_METHOD

METHOD PRIVATE ParseRecvPayloadSequence
VAR_IN_OUT
  /// Robot assignment of function
  AxesGroup        : AxesGroup;
END_VAR

VAR
  /// internal index
 _idx              : DINT;
  /// index for sequence
 _seqIdx           : DINT;
  /// index for fragment
 _fragIdx          : DINT; 
  /// current payload pointer for current fragment
 _payLoadPtr       : DINT;
  /// Amount of sequences
 _seqCount         : DINT;
  /// current payload pointer of the current sequence
 _seqPayloadPtr    : UINT; 
END_VAR
                  // Check 2nd sequence active ? 
IF ( _parCfg.Com.TwoSequences )
THEN
 _seqCount := _seqCount + 1;
END_IF

FOR _seqIdx := 0 TO _seqCount
DO
  // Check 2nd sequence ? -> goto 2nd sequence payload address  
  IF ( _seqIdx = SECONDARY_SEQUENCE )
  THEN
    RecvData.PayloadPtr := CalculateSequencePayloadStartAdr(AxesGroup := AxesGroup, 
                                                            Direction := ComDirection.ROB_TO_PLC,
                                                            Sequence  := SequenceFlag.SECONDARY_SEQUENCE);
	END_IF

  // parste sequence header
  Telegram.RobToPlc.Sequence[_seqIdx].Header.SEQ_ACK       := RecvData.GetUint();
  Telegram.RobToPlc.Sequence[_seqIdx].Header.PayloadLength := RecvData.GetUint();
  
  // check new data available ? 
  IF ( Telegram.RobToPlc.Sequence[_seqIdx].Header.SEQ_ACK <> AxesGroup.State.LastACK[_seqIdx]) 
  THEN
    // Check sequence payload available ? 
    IF (Telegram.RobToPlc.Sequence[_seqIdx].Header.PayloadLength > 0)
    THEN
      // Check sequence payload length is valid ? 
      IF ( Telegram.RobToPlc.Sequence[_seqIdx].Header.PayloadLength > _parCfg.Com.TelegramLengthRobToPlc )
      THEN 
        // Create log entry for payload not valid 
        CreateLogMessagePara2 ( Timestamp   := SystemTime,
                                MessageType := MessageType.CMD,
                                Severity    := Severity.DEBUG,
                                MessageCode := 0,
                                MessageText := 'Invalid sequence payload length, Sequence = {1}, PayloadLength = {2} ',
                                Para1       :=  DINT_TO_STRING(_seqIdx),
                                Para2       :=  UINT_TO_STRING(Telegram.RobToPlc.Sequence[_seqIdx].Header.PayloadLength));
                                RETURN;
      ELSE
        // Create log entry
        CreateLogMessagePara4 ( Timestamp   := SystemTime,
                                MessageType := MessageType.CMD,
                                Severity    := Severity.DEBUG,
                                MessageCode := 0,
                                MessageText := 'RecvData: ACK = {1}, received Sequence [{2}] with PayloadLength = {3}, Lifesign = {4}',
                                Para1       :=  UINT_TO_STRING(Telegram.RobToPlc.Sequence[_seqIdx].Header.SEQ_ACK),
                                Para2       :=  DINT_TO_STRING(_seqIdx),
                                Para3       :=  UINT_TO_STRING(Telegram.RobToPlc.Sequence[_seqIdx].Header.PayloadLength),
                                Para4       :=  BYTE_TO_STRING(Telegram.RobToPlc.Header.LifeSign));
      END_IF
    
      // processing sequence payload                                  
      WHILE ( _seqPayloadPtr < Telegram.RobToPlc.Sequence[_seqIdx].Header.PayloadLength )
      DO                        
        // parse header
        Telegram.RobToPlc.Sequence[_seqIdx].Fragment[_fragIdx].Header.CmdID          := RecvData.GetUint();
        Telegram.RobToPlc.Sequence[_seqIdx].Fragment[_fragIdx].Header.Reserve        := RecvData.GetByte();
        Telegram.RobToPlc.Sequence[_seqIdx].Fragment[_fragIdx].Header.FragmentAction := RecvData.GetByte();
        Telegram.RobToPlc.Sequence[_seqIdx].Fragment[_fragIdx].Header.PayloadPointer := RecvData.GetUint();
        Telegram.RobToPlc.Sequence[_seqIdx].Fragment[_fragIdx].Header.PayloadLength  := RecvData.GetUint();
       
        // add header size to payload pointer 
       _seqPayloadPtr := _seqPayloadPtr + SIZEOF(Telegram.RobToPlc.Sequence[_seqIdx].Fragment[_fragIdx].Header);
        
        // Check fragment payload available ? 
        IF (Telegram.RobToPlc.Sequence[_seqIdx].Fragment[_fragIdx].Header.PayloadLength > 0)
        THEN
          // Check fragment payload length is valid ? 
          IF ( Telegram.RobToPlc.Sequence[_seqIdx].Fragment[_fragIdx].Header.PayloadLength > _parCfg.Com.TelegramLengthRobToPlc )
          THEN 
            // Create log entry for payload not valid 
            CreateLogMessagePara2 ( Timestamp   := SystemTime,
                                    MessageType := MessageType.CMD,
                                    Severity    := Severity.DEBUG,
                                    MessageCode := 0,
                                    MessageText := 'Invalid fragment payload length, Sequence = {1}, PayloadLength = {2} ',
                                    Para1       :=  DINT_TO_STRING(_seqIdx),
                                    Para2       :=  UINT_TO_STRING(Telegram.RobToPlc.Sequence[_seqIdx].Fragment[_fragIdx].Header.PayloadLength));
                                    RETURN;
          END_IF
        
          // Fill Response payload
          FOR _idx := 0 TO Telegram.RobToPlc.Sequence[_seqIdx].Fragment[_fragIdx].Header.PayloadLength -1
          DO
            // calculate payload pointer
           _payLoadPtr := Telegram.RobToPlc.Sequence[_seqIdx].Fragment[_fragIdx].Header.PayloadPointer + _idx;
          
            IF (( _payLoadPtr >= 0                                          ) AND
                ( _payLoadPtr <= RobotLibraryParameter.RESPONSE_PAYLOAD_MAX ))
            THEN  
              Telegram.RobToPlc.Sequence[_seqIdx].Fragment[_fragIdx].Command.Payload[_payLoadPtr] := RecvData.GetByte();
              // inc payload pointer
             _seqPayloadPtr := _seqPayloadPtr + SIZEOF(BYTE);
            ELSE
              // Create log entry for payload pointer not valid 
              CreateLogMessagePara3 ( Timestamp   := SystemTime,
                                      MessageType := MessageType.CMD,
                                      Severity    := Severity.DEBUG,
                                      MessageCode := 0,
                                      MessageText := 'Invalid fragment payload pointer, Sequence = {1}, Fragment = {2}, PayloadPointer = {3} ',
                                      Para1       :=  DINT_TO_STRING(_seqIdx),
                                      Para2       :=  DINT_TO_STRING(_fragIdx),
                                      Para3       :=  DINT_TO_STRING(_payLoadPtr));
                                      RETURN;
					  END_IF
           
          END_FOR
          
          // Add Response to ACR
          AxesGroup.Acyclic.ActiveCommandRegister.AddRsp(Telegram.RobToPlc.Sequence[_seqIdx].Fragment[_fragIdx]);
        
          // Only for debugging - header is part of the payload itself
          Telegram.RobToPlc.Sequence[_seqIdx].Fragment[_fragIdx].Command.Header.State                 :=      GetHalfeByteLo( Value :=  Telegram.RobToPlc.Sequence[_seqIdx].Fragment[_fragIdx].Command.Payload[0]);
          Telegram.RobToPlc.Sequence[_seqIdx].Fragment[_fragIdx].Command.Header.ParSeq                :=      GetHalfeByteHi( Value :=  Telegram.RobToPlc.Sequence[_seqIdx].Fragment[_fragIdx].Command.Payload[0]);
          Telegram.RobToPlc.Sequence[_seqIdx].Fragment[_fragIdx].Command.Header.AlarmMessageSeverity  :=        BYTE_TO_SINT(           Telegram.RobToPlc.Sequence[_seqIdx].Fragment[_fragIdx].Command.Payload[1]);
          Telegram.RobToPlc.Sequence[_seqIdx].Fragment[_fragIdx].Command.Header.AlarmMessageCode      :=  CombineBytesToUint( HiByte := Telegram.RobToPlc.Sequence[_seqIdx].Fragment[_fragIdx].Command.Payload[2],
                                                                                                                              LoByte := Telegram.RobToPlc.Sequence[_seqIdx].Fragment[_fragIdx].Command.Payload[3]);
          // Create log entry
          CreateLogMessagePara5 ( Timestamp   := SystemTime,
                                  MessageType := MessageType.CMD,
                                  Severity    := Severity.DEBUG,
                                  MessageCode := 0,
                                  MessageText := 'RecvData: received Fragment [{1}] with PayloadLength = {2}, CmdID <{3}> , CmdState: {4}, Fragment-Action Bits: {5}',
                                  Para1       :=  DINT_TO_STRING(_seqIdx),
                                  Para2       :=  UINT_TO_STRING              (Telegram.RobToPlc.Sequence[_seqIdx].Fragment[_fragIdx].Header.PayloadLength),
                                  Para3       :=  DINT_TO_STRING              (Telegram.RobToPlc.Sequence[_seqIdx].Fragment[_fragIdx].Header.CmdID),
                                  Para4       :=  CMD_MESSAGE_STATE_TO_STRING (Telegram.RobToPlc.Sequence[_seqIdx].Fragment[_fragIdx].Command.Header.State),
                                  Para5       :=    FRAGMENT_ACTION_TO_STRING (Telegram.RobToPlc.Sequence[_seqIdx].Fragment[_fragIdx].Header.FragmentAction));
        END_IF
        
        // Check still payload left ? -> goto next fragment  
        IF ( _seqPayloadPtr < Telegram.RobToPlc.Sequence[_seqIdx].Header.PayloadLength )
        THEN
         _fragIdx := _fragIdx + 1;        
        END_IF
        
        // Check fragment index limit reached ? 
        IF ( _fragIdx > RobotLibraryParameter.FRAGMENT_MAX ) 
        THEN 
          // Create log entry
          CreateLogMessagePara1 ( Timestamp   := SystemTime,
                                  MessageType := MessageType.CMD,
                                  Severity    := Severity.DEBUG,
                                  MessageCode := 0,
                                  MessageText := 'Fragment index out of range, _fragIdx = {1} ',
                                  Para1       :=  DINT_TO_STRING(_fragIdx));
                                  RETURN;
        END_IF        
      END_WHILE    
    END_IF
  END_IF    
END_FOR  
                
END_METHOD

METHOD Reset
VAR_IN_OUT
  /// Robot assignment of function
  AxesGroup : AxesGroup;  
END_VAR
                  // reset flags
Busy              := FALSE;
Initialized       := FALSE;
Synchronized      := FALSE;
Error             := FALSE;
ErrorID           := 0;
ErrorAddTxt       := '';
WarningID         := 0;
InfoID            := 0;  

// Reset internal functon blocks
_exchangeConfiguration      .Enable  := FALSE;
_readRobotData              .Execute := FALSE;
_readMessages               .Enable  := FALSE;  
_readToolData               .Execute := FALSE;  
_readFrameData              .Execute := FALSE;  
_readLoadData               .Execute := FALSE;  
_readWorkArea               .Execute := FALSE;  
_readRobotSWLimits          .Execute := FALSE;  
_readRobotDefaultDynamics   .Execute := FALSE;  
_readRobotReferenceDynamics .Execute := FALSE;  
_writeToolData              .Execute := FALSE;   
_writeFrameData             .Execute := FALSE;   
_writeLoadData              .Execute := FALSE;   
_writeWorkArea              .Execute := FALSE;   
_writeRobotSWLimits         .Execute := FALSE;   
_writeRobotDefaultDynamics  .Execute := FALSE;   
_writeRobotReferenceDynamics.Execute := FALSE;   

// Set Client error to force server error
AxesGroup.Cyclic.PlcToRob.Control := ControlHalfByte.NONE;

// Reset synchronisation state variables
AxesGroup.State.SyncStatePlc.InSync.Frame             := FALSE;
AxesGroup.State.SyncStatePlc.InSync.Tool              := FALSE;
AxesGroup.State.SyncStatePlc.InSync.Load              := FALSE;
AxesGroup.State.SyncStatePlc.InSync.WorkArea          := FALSE;
AxesGroup.State.SyncStatePlc.InSync.SwLimits          := FALSE;
AxesGroup.State.SyncStatePlc.InSync.DefaultDynamics   := FALSE;
AxesGroup.State.SyncStatePlc.InSync.ReferenceDynamics := FALSE;

AxesGroup.State.SyncStatePlc.UnSyncNo.Frame    := 0;
AxesGroup.State.SyncStatePlc.UnSyncNo.Tool     := 0;
AxesGroup.State.SyncStatePlc.UnSyncNo.Load     := 0;
AxesGroup.State.SyncStatePlc.UnSyncNo.WorkArea := 0;

AxesGroup.State.SyncStateRc .InSync.Frame             := FALSE;
AxesGroup.State.SyncStateRc .InSync.Tool              := FALSE;
AxesGroup.State.SyncStateRc .InSync.Load              := FALSE;
AxesGroup.State.SyncStateRc .InSync.WorkArea          := FALSE;
AxesGroup.State.SyncStateRc .InSync.SwLimits          := FALSE;
AxesGroup.State.SyncStateRc .InSync.DefaultDynamics   := FALSE;
AxesGroup.State.SyncStateRc .InSync.ReferenceDynamics := FALSE;

AxesGroup.State.SyncStateRc .UnSyncNo.Frame    := 0;
AxesGroup.State.SyncStateRc .UnSyncNo.Tool     := 0;
AxesGroup.State.SyncStateRc .UnSyncNo.Load     := 0;
AxesGroup.State.SyncStateRc .UnSyncNo.WorkArea := 0;

// Reset active command register
AxesGroup.Acyclic.ActiveCommandRegister.Reset();
      
// reset step counters
_stepCmd                   := 0;
_stepSyncFrameData         := 0;
_stepSyncLoadData          := 0;
_stepSyncDefaultDynamics   := 0;
_stepSyncReferenceDynamics := 0;
_stepSyncSWLimits          := 0;
_stepSyncToolData          := 0;
_stepSyncWorkArea          := 0;
                
END_METHOD

METHOD PUBLIC SetError
VAR_INPUT
  /// ErrorID reported by RC for error identification according to Table 7-1
  ErrorID   : WORD;
  /// TRUE = overwrite an existing error 
  Overwrite : BOOL;
END_VAR
                  IF ( NOT HasError ) OR ( Overwrite )
THEN
  THIS^.ErrorID := ErrorID;
END_IF
                
END_METHOD

METHOD PUBLIC SetInfo
VAR_INPUT
  /// InfoID for info identification reported during execution of command according to Table 7-5
  InfoID    : WORD;
  /// TRUE = overwrite an existing info 
  Overwrite : BOOL;
END_VAR
                  IF ( NOT HasInfo ) OR ( Overwrite )
THEN
  THIS^.InfoID := InfoID;
END_IF
                
END_METHOD

METHOD PUBLIC SetWarning
VAR_INPUT
  /// WarningID for warning identification reported during execution of command according to Table 7-3
  WarningID : WORD;
  /// TRUE = overwrite an existing warning 
  Overwrite : BOOL;
END_VAR
                  IF ( NOT HasWarning ) OR ( Overwrite )
THEN
  THIS^.WarningID := WarningID;
END_IF
                
END_METHOD

PROPERTY PROTECTED HasError : Bool
GET
VAR
END_VAR
                    HasError := ErrorID <> RobotLibraryErrorIdEnum.NO_ERROR;
                  
END_GET
END_PROPERTY

PROPERTY PROTECTED HasInfo : BOOL
GET
VAR
END_VAR
                    HasInfo := InfoID <> RobotLibraryInfoIdEnum.NO_INFO;
                  
END_GET
END_PROPERTY

PROPERTY PROTECTED HasWarning : BOOL
GET
VAR
END_VAR
                    HasWarning := WarningID <> RobotLibraryWarningIdEnum.NO_WARNING;
                  
END_GET
END_PROPERTY
END_FUNCTION_BLOCK

/// Switch operation mode of RC (Automatic External, T1 External, T2 External)
FUNCTION_BLOCK MC_SetOperationModeFB EXTENDS RobotLibraryBaseExecuteFB
// ------------------------------------------------------------------------- 
//  SRCI Robot Library                                                
// ------------------------------------------------------------------------- 
//                                                                           
//  Object:      SetOperationModeFB                                       
//  Author:      Thorsten Brach                                                
//  Date:        2024-06-01
//
//  Description:                                              
//   
//                                                                           
//  Copyright: 
//    (C) 2024 Thorsten Brach. All rights reserved                                                                                                                                            
//             Licensed under the MIT License.
//                                                                           
//  Disclaimer:                                                                           
//    This project is provided without any guarantee and can be used for   
//    private and commercial purposes. Any use is at the user’s 
//    own risk and responsibility.
//
// -------------------------------------------------------------------------
VAR_INPUT
  /// command parameter 
  ParCmd          : SetOperationModeParCmd;
END_VAR
VAR_OUTPUT
  /// Command is transferred and confirmed by the RC
  CommandBuffered : BOOL;
  /// command results
  OutCmd          : SetOperationModeOutCmd;     
END_VAR

VAR
  /// internal copy of command parameter 
 _parCmd          : SetOperationModeParCmd;
  /// command data to send
 _command         : SetOperationModeSendData;
  /// response data received
 _response        : SetOperationModeRecvData;      
END_VAR

            SUPER^(AxesGroup := AxesGroup);
          

METHOD INTERNAL CheckAddParameter : BOOL
VAR_INPUT
  /// Payload pointer
  PayloadPtr : UDINT;
END_VAR
VAR
  /// Payload as byte array
  Payload    : ARRAY [1..SIZEOF(_command)] OF BYTE;
  /// Null Byte array 
  Null       : ARRAY [1..SIZEOF(_command)] OF BYTE;
  /// Data length to compare
  DataLen    : UDINT;
END_VAR
                  // Payload pointer must be decreased by one byte, because ADR(Payload) is already one byte !
PayloadPtr := LIMIT (0, PayloadPtr - 1, SIZEOF(Payload) -1);
// Convert command struct to payload array
SysDepMemCpy( pDest := ADR(Payload), pSrc := ADR(_command), DataLen := SIZEOF(_command));
// Calculate the data length to compare - at least one byte must be compared !
DataLen := LIMIT(1, SIZEOF(Payload) - PayloadPtr, SIZEOF(Payload)); 
// Compare Payload-Array with Null-Byte-Array
CheckAddParameter := SysDepMemCmp( pData1 := ADR(Payload) + PayloadPtr , pData2 := ADR(Null), DataLen := DataLen) <>  RobotLibraryConstants.OK ;
                
END_METHOD

METHOD PROTECTED CheckFunctionSupported : BOOL
VAR_IN_OUT
  /// Robot assignment of function
  AxesGroup : AxesGroup; 
END_VAR
                  CheckFunctionSupported := AxesGroup.State.RobotData.RCSupportedFunctions.SetOperationMode;

IF ( NOT CheckFunctionSupported )
THEN
  // call base implementation for set error and create log entry
  SUPER^.CheckFunctionSupported(AxesGroup := AxesGroup);
END_IF
                
END_METHOD

METHOD PROTECTED CheckParameterChanged : BOOL
VAR_IN_OUT
  /// Robot assignment of function
  AxesGroup    : AxesGroup; 
END_VAR
                  // Check ParCmd Size is > 0, because MemCmp does not work correctly with size = 0
IF (SIZEOF(ParCmd) = 0) OR (_stepCmd = 0)
THEN 
  RETURN;
END_IF

// compare memory 
_parameterChanged := ( SysDepMemCmp(pData1 := ADR(ParCmd), pData2 := ADR(_parCmd), DataLen := SIZEOF(ParCmd)) <> RobotLibraryConstants.OK );

// check parameter valid ?
_parameterValid   := CheckParameterValid( AxesGroup := AxesGroup );

IF ((  _parameterChanged        )  AND 
    (  _parameterValid          )) OR
    (  _parameterUpdateInternal )  
THEN  
  // Create log entry for parameter changed event
  CreateLogMessagePara1 ( Timestamp   := AxesGroup.State.SystemTime,
                          MessageType := MessageType.CMD,
                          Severity    := Severity.DEBUG,
                          MessageCode := 0,
                          MessageText := 'NotifyParameterChanged Event {1}',
                          Para1       :=  '' );

  // reset internal flag for send parameter update
 _parameterUpdateInternal := FALSE;
  // update internal copy of parameters 
 _parCmd := ParCmd;
  // inc parameter sequence
 _command.ParSeq := _command.ParSeq + 1;
  // update command data  
  CommandData := CreateCommandPayload(AxesGroup := AxesGroup); // ( Access via reference to rCommandFB in ACR )
  // notify active command register 
  AxesGroup.Acyclic.ActiveCommandRegister.NotifyParameterChanged := _uniqueID;
END_IF
                
END_METHOD

METHOD PROTECTED CheckParameterValid : BOOL
VAR_IN_OUT
  /// Robot assignment of function
  AxesGroup : AxesGroup; 
END_VAR
VAR
  /// internal index for loops
 _idx : DINT;
END_VAR
                  CheckParameterValid := TRUE;

// Check ParCmd.OperationMode valid ? 
IF (( ParCmd.OperationMode <> OperationMode.AUTO_EXT ) AND  
    ( ParCmd.OperationMode <> OperationMode.T1_EXT   ) AND  
    ( ParCmd.OperationMode <> OperationMode.T2_EXT   ))  
THEN
  // Parameter not valid
  CheckParameterValid := FALSE;
  // Set error
  SetError( ErrorID := RobotLibraryErrorIdEnum.ERR_INVALID_PAR_CMD, Overwrite := TRUE );
  // Create log entry
  CreateLogMessagePara1 ( Timestamp   := AxesGroup.State.SystemTime,
                          MessageType := MessageType.CMD,
                          Severity    := Severity.ERROR,
                          MessageCode := ErrorID,
                          MessageText := 'Invalid Parameter ParCmd.OperationMode = {1}',
                          Para1       :=  OPERATION_MODE_TO_STRING(ParCmd.OperationMode));
  RETURN;                          
END_IF

                
END_METHOD

METHOD INTERNAL CreateCommandPayload : RobotLibraryCommandDataFB
VAR_IN_OUT
  /// Robot assignment of function
  AxesGroup : AxesGroup; 
END_VAR
VAR
  /// Parameter count
 _parameterCnt : DINT;
END_VAR
// Table 6-193: Sent CMD payload (PLC to RC) of "SetOperationMode"
// --------------------------
// Header
// --------------------------
// Byte 00 : UINT  - Type HB     
// Byte 01 :       - Type LB    
// Byte 02 : USINT - Reserve | ExecutionMode
// Byte 03 : USINT - ParSeq  | Priority
// --------------------------
// Datablock
// --------------------------
 // Byte 04 : UINT  OperationMode;
 // Byte 05 :       OperationMode;
// --------------------------
                  // set command parameter 
_command.CmdTyp        :=  CmdType.SetOperationMode;
_command.ExecMode      :=  ExecMode;
_command.ParSeq        := _command.ParSeq;
_command.Priority      :=  Priority;
_command.OperationMode := _parCmd.OperationMode;

// copy command data to header
_cmdHeader := _command;
// call base implementation to copy header to payload buffer
CreateCommandPayload := SUPER^.CreateCommandPayload(AxesGroup := AxesGroup);


// Check parameter must be added ? 
IF ( CheckAddParameter(CreateCommandPayload.PayloadPtr))
THEN
  // add command.OperationMode
  CreateCommandPayload.AddUsint(_command.OperationMode);
  // inc parameter counter
 _parameterCnt := _parameterCnt + 1;  
END_IF


// Create logging
CreateCommandPayloadLog(AxesGroup := AxesGroup, ParameterCnt := _parameterCnt);
                
END_METHOD

METHOD INTERNAL CreateCommandPayloadLog 
VAR_IN_OUT
  /// Robot assignment of function
  AxesGroup : AxesGroup; 
END_VAR
VAR_INPUT
  /// Parameter count
  ParameterCnt : DINT;
END_VAR
                  // Create log entry for Parameter start
CreateLogMessagePara1 ( Timestamp   := AxesGroup.State.SystemTime,
                        MessageType := MessageType.CMD,
                        Severity    := Severity.DEBUG,
                        MessageCode := 0,
                        MessageText := 'Create command payload with {1} parameter(s) :',
                        Para1       := DINT_TO_STRING(ParameterCnt));


// Return if no parameter is remaining...
IF ( ParameterCnt = 0 ) THEN RETURN; END_IF
// dec remaining parameter(s)                        
ParameterCnt := ParameterCnt - 1;
// Create log entry for OperationMode
CreateLogMessagePara1 ( Timestamp   := AxesGroup.State.SystemTime,
                        MessageType := MessageType.CMD,
                        Severity    := Severity.DEBUG,
                        MessageCode := 0,
                        MessageText := 'Command.OperationMode = {1}',
                        Para1       :=  USINT_TO_STRING(_command.OperationMode));
                
END_METHOD

METHOD FB_init : BOOL
VAR_INPUT
  /// if TRUE, the retain variables are initialized (warm start / cold start)
  bInitRetains : BOOL; 
  /// if TRUE, the instance afterwards gets moved into the copy code (online change)
  bInCopyCode  : BOOL;  
END_VAR
                  MyType := 'MC_SetOperationModeFB';

ExecMode := ExecutionMode.PARALLEL;
Priority := PriorityLevel.NORMAL;
                
END_METHOD

METHOD PROTECTED OnExecRun : DINT
VAR_IN_OUT
  /// Robot assignment of function
  AxesGroup : AxesGroup; 
END_VAR
                  // call base implementation
SUPER^.OnExecRun(AxesGroup := AxesGroup);

CASE _stepCmd OF
  
  00:  IF ( _execute_R.Q ) AND ( NOT Error) 
       THEN
         // Check function is supported and parameter are valid ?
         IF (( CheckFunctionSupported( AxesGroup := AxesGroup )) AND
             ( CheckParameterValid   ( AxesGroup := AxesGroup )))      
         THEN
           // set busy flag
           Busy := TRUE;
           // Reset command outputs
           SysDepMemSet(pDest := ADR(OutCmd), Value := 0, DataLen := SIZEOF(OutCmd));         
           // apply command parameter
          _parCmd := ParCmd;
           // init parameter sequence
          _command.ParSeq := 1;
           // create command data
           CommandData := CreateCommandPayload(AxesGroup := AxesGroup);
           // Add command to active command register
          _uniqueID := AxesGroup.Acyclic.ActiveCommandRegister.AddCmd( pCommandFB := ADR(THIS^ ));     
           // set timeout
           SetTimeout(PT := _timeoutCmd, rTimer := _timerCmd);
           // inc step counter
          _stepCmd := _stepCmd + 1;
         END_IF 
       END_IF
     

  01:  // Wait for responce received
       IF ( _responseReceived )
       THEN
         // reset response received flag
        _responseReceived := FALSE;
         // update state flags
         OnUpdateStateFlags(_response.State);
         // update state flags
         OnApplyOutCmd(_response.State);

         // Done, Aborted or Error ?
         IF (_response.State >= CmdMessageState.DONE )
         THEN
           // set timeout
           SetTimeout(PT := _timeoutCmd, rTimer := _timerCmd);
           // inc step counter
          _stepCmd := _stepCmd + 1; 
         END_IF
       END_IF


  02: IF ( NOT Execute)
      THEN
        Reset();  
      END_IF     

ELSE
  // invalid step
  SetError( ErrorID := RobotLibraryErrorIdEnum.ERR_INVALID_STEP, Overwrite := TRUE );
END_CASE


// Reset FB
IF ( NOT Execute )
THEN
  Reset(); 
END_IF
                
END_METHOD

METHOD PROTECTED OnUpdateStateFlags
VAR_INPUT
  /// Command message state
  State : CmdMessageState;
END_VAR
                  // Reset State flags
Done := FALSE;

CASE State OF

  // No operation or process is active
  CmdMessageState.EMPTY               :;
  // Created but not yet started
  CmdMessageState.CREATED             :;
  // Buffered and awaiting execution
  CmdMessageState.BUFFERED            : CommandBuffered    := TRUE;
  // Buffered in planner for future execution
  CmdMessageState.BUFFERED_IN_PLANNER : CommandBuffered    := TRUE;
  // Currently active and in progress
  CmdMessageState.ACTIVE              :;                                         
  // Interrupted and awaiting continuation
  CmdMessageState.INTERRUPTED         :;  
  // Requested for abort
  CmdMessageState.ABORT_REQUEST       :;
  // Successfully completed
  CmdMessageState.DONE                : Done               := TRUE;
                                        Busy               := FALSE;
  // Aborted before completion
  CmdMessageState.ABORTED             : Busy               := FALSE;
  // Encountered an error during execution
  CmdMessageState.ERROR               : Error              := TRUE;
                                        Busy               := FALSE;
END_CASE
                
END_METHOD

METHOD INTERNAL ParseResponsePayload : DINT
VAR_INPUT
  /// Response data
  ResponseData : RobotLibraryResponseDataFB;
  /// Timestamp
  Timestamp    : SystemTime;  
END_VAR
VAR
  /// Parameter count
 _parameterCnt : DINT;
END_VAR
// Table 6-194: Received CMD payload (RC to PLC) of "SetOperationMode"
// --------------------------
// Header
// --------------------------
// Byte 00 : USINT   - ParSeq | State     
// Byte 01 : SINT    - AlarmMessageSeverity    
// Byte 02 : UINT    - AlarmMessageCode HB
// Byte 03 :         - AlarmMessageCode LB
// --------------------------
                  // call base implementation to parse the header from payload buffer
ResponseData.PayloadPtr := SUPER^.ParseResponsePayload(ResponseData := ResponseData, Timestamp := Timestamp);

// copy parsed header to response
_response.ParSeq               := _rspHeader.ParSeq;
_response.State                := _rspHeader.State;
_response.AlarmMessageSeverity := _rspHeader.AlarmMessageSeverity;
_response.AlarmMessageCode     := _rspHeader.AlarmMessageCode;

// Create logging
ParseResponsePayloadLog(ResponseData := ResponseData, Timestamp := Timestamp, ParameterCnt := _parameterCnt);
                
END_METHOD

METHOD INTERNAL ParseResponsePayloadLog
VAR_INPUT
  /// Response data
  ResponseData : RobotLibraryResponseDataFB;
  /// Timestamp
  Timestamp    : SystemTime;  
  /// Parameter count
  ParameterCnt : DINT;
END_VAR
                  // Create log entry for Parameter start
CreateLogMessagePara1 ( Timestamp   := Timestamp,
                        MessageType := MessageType.CMD,
                        Severity    := Severity.DEBUG,
                        MessageCode := 0,
                        MessageText := '{1} parameter(s) to parse from the response data:',
                        Para1       := DINT_TO_STRING(ParameterCnt));
                        

// Return if no parameter is remaining...
IF ( ParameterCnt = 0 ) THEN RETURN; END_IF
// dec remaining parameter(s)                        
ParameterCnt := ParameterCnt - 1;
// Create log entry for no parameter 
CreateLogMessage      ( Timestamp   := Timestamp,
                        MessageType := MessageType.CMD,
                        Severity    := Severity.DEBUG,
                        MessageCode := 0,
                        MessageText := 'This command has no parameter to parse...');
                
END_METHOD

METHOD PROTECTED Reset : DINT
VAR_INPUT
END_VAR
                  Reset := SUPER^.Reset();

Done               := FALSE;
Busy               := FALSE;
CommandBuffered    := FALSE;
                
END_METHOD
END_FUNCTION_BLOCK

/// Set active sequence
FUNCTION_BLOCK MC_SetSequenceFB EXTENDS RobotLibraryBaseExecuteFB
// ------------------------------------------------------------------------- 
//  SRCI Robot Library                                                
// ------------------------------------------------------------------------- 
//                                                                           
//  Object:      SetSequenceFB                                       
//  Author:      Thorsten Brach                                                
//  Date:        2024-06-01
//
//  Description:                                              
//   
//                                                                           
//  Copyright: 
//    (C) 2024 Thorsten Brach. All rights reserved                                                                                                                                            
//             Licensed under the MIT License.
//                                                                           
//  Disclaimer:                                                                           
//    This project is provided without any guarantee and can be used for   
//    private and commercial purposes. Any use is at the user’s 
//    own risk and responsibility.
//
// -------------------------------------------------------------------------
VAR_INPUT
  /// command parameter 
  ParCmd          : SetSequenceParCmd;  
END_VAR

VAR_OUTPUT
  /// Command is transferred and confirmed by the RC
  CommandBuffered : BOOL;
  /// command results
  OutCmd          : SetSequenceOutCmd;     
END_VAR

VAR
  /// internal copy of command parameter 
 _parCmd          : SetSequenceParCmd;
  /// command data to send
 _command         : SetSequenceSendData;
  /// response data received
 _response        : SetSequenceRecvData;      
END_VAR

            SUPER^(AxesGroup := AxesGroup);
          

METHOD INTERNAL CheckAddParameter : BOOL
VAR_INPUT
  /// Payload pointer
  PayloadPtr : UDINT;
END_VAR
VAR
  /// Payload as byte array
  Payload    : ARRAY [1..SIZEOF(_command)] OF BYTE;
  /// Null Byte array 
  Null       : ARRAY [1..SIZEOF(_command)] OF BYTE;
  /// Data length to compare
  DataLen    : UDINT;
END_VAR
                  // Payload pointer must be decreased by one byte, because ADR(Payload) is already one byte !
PayloadPtr := LIMIT (0, PayloadPtr - 1, SIZEOF(Payload) -1);
// Convert command struct to payload array
SysDepMemCpy( pDest := ADR(Payload), pSrc := ADR(_command), DataLen := SIZEOF(_command));
// Calculate the data length to compare - at least one byte must be compared !
DataLen := LIMIT(1, SIZEOF(Payload) - PayloadPtr, SIZEOF(Payload)); 
// Compare Payload-Array with Null-Byte-Array
CheckAddParameter := SysDepMemCmp( pData1 := ADR(Payload) + PayloadPtr , pData2 := ADR(Null), DataLen := DataLen) <>  RobotLibraryConstants.OK ;
                
END_METHOD

METHOD PROTECTED CheckFunctionSupported : BOOL
VAR_IN_OUT
  /// Robot assignment of function
  AxesGroup : AxesGroup; 
END_VAR
                  CheckFunctionSupported := AxesGroup.State.RobotData.RCSupportedFunctions.SetSequence;

IF ( NOT CheckFunctionSupported )
THEN
  // call base implementation for set error and create log entry
  SUPER^.CheckFunctionSupported(AxesGroup := AxesGroup);
END_IF
                
END_METHOD

METHOD PROTECTED CheckParameterChanged : BOOL
VAR_IN_OUT
  /// Robot assignment of function
  AxesGroup    : AxesGroup; 
END_VAR
                  // Check ParCmd Size is > 0, because MemCmp does not work correctly with size = 0
IF (SIZEOF(ParCmd) = 0) OR (_stepCmd = 0)
THEN 
  RETURN;
END_IF

// compare memory 
_parameterChanged := ( SysDepMemCmp(pData1 := ADR(ParCmd), pData2 := ADR(_parCmd), DataLen := SIZEOF(ParCmd)) <> RobotLibraryConstants.OK );

// check parameter valid ?
_parameterValid   := CheckParameterValid( AxesGroup := AxesGroup );

IF ((  _parameterChanged        )  AND 
    (  _parameterValid          )) OR
    (  _parameterUpdateInternal )  
THEN  
  // Create log entry for parameter changed event
  CreateLogMessagePara1 ( Timestamp   := AxesGroup.State.SystemTime,
                          MessageType := MessageType.CMD,
                          Severity    := Severity.DEBUG,
                          MessageCode := 0,
                          MessageText := 'NotifyParameterChanged Event {1}',
                          Para1       :=  '' );

  // reset internal flag for send parameter update
 _parameterUpdateInternal := FALSE;
  // update internal copy of parameters 
 _parCmd := ParCmd;
  // inc parameter sequence
 _command.ParSeq := _command.ParSeq + 1;
  // update command data  
  CommandData := CreateCommandPayload(AxesGroup := AxesGroup); // ( Access via reference to rCommandFB in ACR )
  // notify active command register 
  AxesGroup.Acyclic.ActiveCommandRegister.NotifyParameterChanged := _uniqueID;
END_IF
                
END_METHOD

METHOD PROTECTED CheckParameterValid : BOOL
VAR_IN_OUT
  /// Robot assignment of function
  AxesGroup : AxesGroup; 
END_VAR
VAR
  /// internal index for loops
 _idx : DINT;
END_VAR
                  CheckParameterValid := TRUE;

// Check ParCmd.OperationMode valid ? 
IF (( ParCmd.TargetSequence <> SequenceFlag.PRIMARY_SEQUENCE   ) AND  
    ( ParCmd.TargetSequence <> SequenceFlag.SECONDARY_SEQUENCE ))  
THEN
  // Parameter not valid
  CheckParameterValid := FALSE;
  // Set error
  SetError( ErrorID := RobotLibraryErrorIdEnum.ERR_INVALID_PAR_CMD, Overwrite := TRUE );
  // Create log entry
  CreateLogMessagePara1 ( Timestamp   := AxesGroup.State.SystemTime,
                          MessageType := MessageType.CMD,
                          Severity    := Severity.ERROR,
                          MessageCode := ErrorID,
                          MessageText := 'Invalid Parameter ParCmd.TargetSequence = {1}',
                          Para1       :=  SEQUENCE_FLAG_TO_STRING(ParCmd.TargetSequence));
  RETURN;                          
END_IF

                
END_METHOD

METHOD INTERNAL CreateCommandPayload : RobotLibraryCommandDataFB
VAR_IN_OUT
  /// Robot assignment of function
  AxesGroup : AxesGroup; 
END_VAR
VAR
  /// Parameter count
 _parameterCnt : DINT;
END_VAR
// Table 6-92: Sent CMD payload (PLC to RC) of "SetSequence"
// --------------------------
// Header
// --------------------------
// Byte 00 : UINT  - Type HB     
// Byte 01 :       - Type LB    
// Byte 02 : USINT - Reserve | ExecutionMode
// Byte 03 : USINT - ParSeq  | Priority
// --------------------------
// Datablock
// --------------------------
// Byte 04 : UINT  TargetSequence;
                  // set command parameter 
_command.CmdTyp         :=  CmdType.SetSequence;
_command.ExecMode       :=  ExecMode;
_command.ParSeq         := _command.ParSeq;
_command.Priority       :=  Priority;
_command.TargetSequence := _parCmd.TargetSequence;

// copy command data to header
_cmdHeader := _command;
// call base implementation to copy header to payload buffer
CreateCommandPayload := SUPER^.CreateCommandPayload(AxesGroup := AxesGroup);

// Check parameter must be added ? 
IF ( CheckAddParameter(CreateCommandPayload.PayloadPtr))
THEN
  // add command.TargetSequence
  CreateCommandPayload.AddUsint(_command.TargetSequence);
  // inc parameter counter
 _parameterCnt := _parameterCnt + 1;  
END_IF

// Create logging
CreateCommandPayloadLog(AxesGroup := AxesGroup, ParameterCnt := _parameterCnt);
                
END_METHOD

METHOD INTERNAL CreateCommandPayloadLog 
VAR_IN_OUT
  /// Robot assignment of function
  AxesGroup : AxesGroup; 
END_VAR
VAR_INPUT
  /// Parameter count
  ParameterCnt : DINT;
END_VAR
                  // Create log entry for Parameter start
CreateLogMessagePara1 ( Timestamp   := AxesGroup.State.SystemTime,
                        MessageType := MessageType.CMD,
                        Severity    := Severity.DEBUG,
                        MessageCode := 0,
                        MessageText := 'Create command payload with {1} parameter(s) :',
                        Para1       := DINT_TO_STRING(ParameterCnt));


// Return if no parameter is remaining...
IF ( ParameterCnt = 0 ) THEN RETURN; END_IF
// dec remaining parameter(s)                        
ParameterCnt := ParameterCnt - 1;
// Create log entry for TargetSequence
CreateLogMessagePara1 ( Timestamp   := AxesGroup.State.SystemTime,
                        MessageType := MessageType.CMD,
                        Severity    := Severity.DEBUG,
                        MessageCode := 0,
                        MessageText := 'Command.TargetSequence = {1}',
                        Para1       :=  USINT_TO_STRING(_command.TargetSequence));
                
END_METHOD

METHOD FB_init : BOOL
VAR_INPUT
  /// if TRUE, the retain variables are initialized (warm start / cold start)
  bInitRetains : BOOL; 
  /// if TRUE, the instance afterwards gets moved into the copy code (online change)
  bInCopyCode  : BOOL;  
END_VAR
                  MyType := 'MC_SetSequenceFB';

ExecMode := ExecutionMode.PARALLEL;
Priority := PriorityLevel.NORMAL;
                
END_METHOD

METHOD PROTECTED OnExecRun : DINT
VAR_IN_OUT
  /// Robot assignment of function
  AxesGroup : AxesGroup; 
END_VAR
                  // call base implementation
SUPER^.OnExecRun(AxesGroup := AxesGroup);

CASE _stepCmd OF
  
  00:  IF ( _execute_R.Q ) AND ( NOT Error)  
       THEN
         // Check function is supported and parameter are valid ?
         IF (( CheckFunctionSupported( AxesGroup := AxesGroup )) AND
             ( CheckParameterValid   ( AxesGroup := AxesGroup )))      
         THEN
           // set busy flag
           Busy := TRUE;
           // Reset command outputs
           SysDepMemSet(pDest := ADR(OutCmd), Value := 0, DataLen := SIZEOF(OutCmd));         
           // apply command parameter
          _parCmd := ParCmd;
           // init parameter sequence
          _command.ParSeq := 1;
           // create command data
           CommandData := CreateCommandPayload(AxesGroup := AxesGroup);
           // Add command to active command register
          _uniqueID := AxesGroup.Acyclic.ActiveCommandRegister.AddCmd( pCommandFB := ADR(THIS^ ));     
           // set timeout
           SetTimeout(PT := _timeoutCmd, rTimer := _timerCmd);
           // inc step counter
          _stepCmd := _stepCmd + 1;
         END_IF 
       END_IF
     

  01:  // Wait for responce received
       IF ( _responseReceived )
       THEN
         // reset response received flag
        _responseReceived := FALSE;
         // update state flags
         OnUpdateStateFlags(_response.State);
         // update state flags
         OnApplyOutCmd(_response.State);
                
         // Done, Aborted or Error ?
         IF (_response.State >= CmdMessageState.DONE )
         THEN
           // set timeout
           SetTimeout(PT := _timeoutCmd, rTimer := _timerCmd);
           // inc step counter
          _stepCmd := _stepCmd + 1; 
         END_IF
       END_IF


  02: IF ( NOT Execute)
      THEN
        Reset();
      END_IF     

ELSE
  // invalid step
  SetError( ErrorID := RobotLibraryErrorIdEnum.ERR_INVALID_STEP, Overwrite := TRUE );
END_CASE


// Reset FB
IF ( NOT Execute )
THEN
  Reset();
END_IF
                
END_METHOD

METHOD PROTECTED OnUpdateStateFlags
VAR_INPUT
  /// Command message state
  State : CmdMessageState;
END_VAR
                  // Reset State flags
Done := FALSE;

CASE State OF

  // No operation or process is active
  CmdMessageState.EMPTY               :;
  // Created but not yet started
  CmdMessageState.CREATED             :;
  // Buffered and awaiting execution
  CmdMessageState.BUFFERED            : CommandBuffered    := TRUE;
  // Buffered in planner for future execution
  CmdMessageState.BUFFERED_IN_PLANNER : CommandBuffered    := TRUE;
  // Currently active and in progress
  CmdMessageState.ACTIVE              :;                                         
  // Interrupted and awaiting continuation
  CmdMessageState.INTERRUPTED         :;  
  // Requested for abort
  CmdMessageState.ABORT_REQUEST       :;
  // Successfully completed
  CmdMessageState.DONE                : Done               := TRUE;
                                        Busy               := FALSE;
  // Aborted before completion
  CmdMessageState.ABORTED             : Busy               := FALSE;
  // Encountered an error during execution
  CmdMessageState.ERROR               : Error              := TRUE;
                                        Busy               := FALSE;
END_CASE
                
END_METHOD

METHOD INTERNAL ParseResponsePayload : DINT
VAR_INPUT
  /// Response data
  ResponseData : RobotLibraryResponseDataFB;
  /// Timestamp
  Timestamp    : SystemTime;  
END_VAR
VAR
  /// Parameter count
 _parameterCnt : DINT;
END_VAR
// Table 6-93: Received CMD payload (RC to PLC) of "SetSequence"
// --------------------------
// Header
// --------------------------
// Byte 00 : USINT   - ParSeq | State     
// Byte 01 : SINT    - AlarmMessageSeverity    
// Byte 02 : UINT    - AlarmMessageCode HB
// Byte 03 :         - AlarmMessageCode LB
                  // call base implementation to parse the header from payload buffer
ResponseData.PayloadPtr := SUPER^.ParseResponsePayload(ResponseData := ResponseData, Timestamp := Timestamp);

// copy parsed header to response
_response.ParSeq               := _rspHeader.ParSeq;
_response.State                := _rspHeader.State;
_response.AlarmMessageSeverity := _rspHeader.AlarmMessageSeverity;
_response.AlarmMessageCode     := _rspHeader.AlarmMessageCode;

// Create logging
ParseResponsePayloadLog(ResponseData := ResponseData, Timestamp := Timestamp, ParameterCnt := _parameterCnt);
                
END_METHOD

METHOD INTERNAL ParseResponsePayloadLog
VAR_INPUT
  /// Response data
  ResponseData : RobotLibraryResponseDataFB;
  /// Timestamp
  Timestamp    : SystemTime;  
  /// Parameter count
  ParameterCnt : DINT;
END_VAR
                  // Create log entry for Parameter start
CreateLogMessagePara1 ( Timestamp   := Timestamp,
                        MessageType := MessageType.CMD,
                        Severity    := Severity.DEBUG,
                        MessageCode := 0,
                        MessageText := '{1} parameter(s) to parse from the response data:',
                        Para1       := DINT_TO_STRING(ParameterCnt));
                        

// Return if no parameter is remaining...
IF ( ParameterCnt = 0 ) THEN RETURN; END_IF
// dec remaining parameter(s)                        
ParameterCnt := ParameterCnt - 1;
// Create log entry for no parameter 
CreateLogMessage      ( Timestamp   := Timestamp,
                        MessageType := MessageType.CMD,
                        Severity    := Severity.DEBUG,
                        MessageCode := 0,
                        MessageText := 'This command has no parameter to parse...');
                
END_METHOD

METHOD PROTECTED Reset : DINT
VAR_INPUT
END_VAR
                  Reset := SUPER^.Reset();

Done               := FALSE;
Busy               := FALSE;
CommandBuffered    := FALSE;
                
END_METHOD
END_FUNCTION_BLOCK

/// Switch language of robot teach pendant from PLC
FUNCTION_BLOCK MC_SwitchLanguageFB EXTENDS RobotLibraryBaseExecuteFB
// ------------------------------------------------------------------------- 
//  SRCI Robot Library                                                
// ------------------------------------------------------------------------- 
//                                                                           
//  Object:      SwitchLanguageFB                                       
//  Author:      Thorsten Brach                                                
//  Date:        2024-06-01
//
//  Description:                                              
//   
//                                                                           
//  Copyright: 
//    (C) 2024 Thorsten Brach. All rights reserved                                                                                                                                            
//             Licensed under the MIT License.
//                                                                           
//  Disclaimer:                                                                           
//    This project is provided without any guarantee and can be used for   
//    private and commercial purposes. Any use is at the user’s 
//    own risk and responsibility.
//
// -------------------------------------------------------------------------
VAR_INPUT
  /// Command parameter 
  ParCmd          : SwitchLanguageParCmd;    
END_VAR

VAR_OUTPUT
  /// Command is transferred and confirmed by the RC
  CommandBuffered : BOOL;
  /// command results
  OutCmd          : SwitchLanguageOutCmd;     
END_VAR

VAR
  /// internal copy of command parameter 
 _parCmd          : SwitchLanguageParCmd;
  /// command data to send
 _command         : SwitchLanguageSendData;
  /// response data received
 _response        : SwitchLanguageRecvData;      
END_VAR

            SUPER^(AxesGroup := AxesGroup);
          

METHOD INTERNAL CheckAddParameter : BOOL
VAR_INPUT
  /// Payload pointer
  PayloadPtr : UDINT;
END_VAR
VAR
  /// Payload as byte array
  Payload    : ARRAY [1..SIZEOF(_command)] OF BYTE;
  /// Null Byte array 
  Null       : ARRAY [1..SIZEOF(_command)] OF BYTE;
  /// Data length to compare
  DataLen    : UDINT;
END_VAR
                  // Payload pointer must be decreased by one byte, because ADR(Payload) is already one byte !
PayloadPtr := LIMIT (0, PayloadPtr - 1, SIZEOF(Payload) -1);
// Convert command struct to payload array
SysDepMemCpy( pDest := ADR(Payload), pSrc := ADR(_command), DataLen := SIZEOF(_command));
// Calculate the data length to compare - at least one byte must be compared !
DataLen := LIMIT(1, SIZEOF(Payload) - PayloadPtr, SIZEOF(Payload)); 
// Compare Payload-Array with Null-Byte-Array
CheckAddParameter := SysDepMemCmp( pData1 := ADR(Payload) + PayloadPtr , pData2 := ADR(Null), DataLen := DataLen) <>  RobotLibraryConstants.OK ;
                
END_METHOD

METHOD PROTECTED CheckFunctionSupported : BOOL
VAR_IN_OUT
  /// Robot assignment of function
  AxesGroup : AxesGroup; 
END_VAR
                  CheckFunctionSupported := AxesGroup.State.RobotData.RCSupportedFunctions.SwitchLanguage;

IF ( NOT CheckFunctionSupported )
THEN
  // call base implementation for set error and create log entry
  SUPER^.CheckFunctionSupported(AxesGroup := AxesGroup);
END_IF
                
END_METHOD

METHOD PROTECTED CheckParameterChanged : BOOL
VAR_IN_OUT
  /// Robot assignment of function
  AxesGroup    : AxesGroup; 
END_VAR
                  // Check ParCmd Size is > 0, because MemCmp does not work correctly with size = 0
IF (SIZEOF(ParCmd) = 0) OR (_stepCmd = 0)
THEN 
  RETURN;
END_IF

// compare memory 
_parameterChanged := ( SysDepMemCmp(pData1 := ADR(ParCmd), pData2 := ADR(_parCmd), DataLen := SIZEOF(ParCmd)) <> RobotLibraryConstants.OK );

// check parameter valid ?
_parameterValid   := CheckParameterValid( AxesGroup := AxesGroup );

IF ((  _parameterChanged        )  AND 
    (  _parameterValid          )) OR
    (  _parameterUpdateInternal )  
THEN  
  // Create log entry for parameter changed event
  CreateLogMessagePara1 ( Timestamp   := AxesGroup.State.SystemTime,
                          MessageType := MessageType.CMD,
                          Severity    := Severity.DEBUG,
                          MessageCode := 0,
                          MessageText := 'NotifyParameterChanged Event {1}',
                          Para1       :=  '' );

  // reset internal flag for send parameter update
 _parameterUpdateInternal := FALSE;
  // update internal copy of parameters 
 _parCmd := ParCmd;
  // inc parameter sequence
 _command.ParSeq := _command.ParSeq + 1;
  // update command data  
  CommandData := CreateCommandPayload(AxesGroup := AxesGroup); // ( Access via reference to rCommandFB in ACR )
  // notify active command register 
  AxesGroup.Acyclic.ActiveCommandRegister.NotifyParameterChanged := _uniqueID;
END_IF
                
END_METHOD

METHOD PROTECTED CheckParameterValid : BOOL
VAR_IN_OUT
  /// Robot assignment of function
  AxesGroup : AxesGroup; 
END_VAR
VAR
  /// internal index for loops
 _idx : DINT;
END_VAR
                  CheckParameterValid := TRUE;


// Check ParCmd.LanguageCode[x] valid ? 
IF ( ParCmd.LanguageCode = '' )  
THEN
  // Parameter not valid
  CheckParameterValid := FALSE;
  // Set error
  SetError( ErrorID := RobotLibraryErrorIdEnum.ERR_INVALID_PAR_CMD, Overwrite := TRUE );
  // Create log entry
  CreateLogMessagePara1 ( Timestamp   := AxesGroup.State.SystemTime,
                          MessageType := MessageType.CMD,
                          Severity    := Severity.ERROR,
                          MessageCode := ErrorID,
                          MessageText := 'Invalid Parameter ParCmd.LanguageCode = {1}',
                          Para1       := ParCmd.LanguageCode);
                       
  RETURN;                          
END_IF
                
END_METHOD

METHOD INTERNAL CreateCommandPayload : RobotLibraryCommandDataFB
VAR_IN_OUT
  /// Robot assignment of function
  AxesGroup : AxesGroup; 
END_VAR
VAR
  /// Parameter count
 _parameterCnt : DINT;
END_VAR
// Table 6-76: Sent CMD payload (PLC to RC) of "SwitchLanguage"
// --------------------------
// Header
// --------------------------
// Byte 00 : UINT  - Type HB     
// Byte 01 :       - Type LB    
// Byte 02 : USINT - Reserve | ExecutionMode
// Byte 03 : USINT - ParSeq  | Priority
// --------------------------
// Datablock
// --------------------------
// Byte 04 : STRING(2)  - LanguageCode[0]
// Byte 05 :            - LanguageCode[1]
                  // set command parameter 
_command.CmdTyp       :=  CmdType.SwitchLanguage;
_command.ExecMode     :=  ExecMode;
_command.ParSeq       := _command.ParSeq;
_command.Priority     :=  Priority;

_command.LanguageCode := _parCmd.LanguageCode;


// copy command data to header
_cmdHeader := _command;
// call base implementation to copy header to payload buffer
CreateCommandPayload := SUPER^.CreateCommandPayload(AxesGroup := AxesGroup);


// Check parameter must be added ? 
IF ( CheckAddParameter(CreateCommandPayload.PayloadPtr))
THEN
  // add command.LanguageCode
  CreateCommandPayload.AddString(_command.LanguageCode);
  // inc parameter counter
 _parameterCnt := _parameterCnt + 1;  
END_IF


// Create logging
CreateCommandPayloadLog(AxesGroup := AxesGroup, ParameterCnt := _parameterCnt);
                
END_METHOD

METHOD INTERNAL CreateCommandPayloadLog 
VAR_IN_OUT
  /// Robot assignment of function
  AxesGroup : AxesGroup; 
END_VAR
VAR_INPUT
  /// Parameter count
  ParameterCnt : DINT;
END_VAR
                  // Create log entry for Parameter start
CreateLogMessagePara1 ( Timestamp   := AxesGroup.State.SystemTime,
                        MessageType := MessageType.CMD,
                        Severity    := Severity.DEBUG,
                        MessageCode := 0,
                        MessageText := 'Create command payload with {1} parameter(s) :',
                        Para1       := DINT_TO_STRING(ParameterCnt));


// Return if no parameter is remaining...
IF ( ParameterCnt = 0 ) THEN RETURN; END_IF
// dec remaining parameter(s)                        
ParameterCnt := ParameterCnt - 1;
// Create log entry for LanguageCode
CreateLogMessagePara1 ( Timestamp   := AxesGroup.State.SystemTime,
                        MessageType := MessageType.CMD,
                        Severity    := Severity.DEBUG,
                        MessageCode := 0,
                        MessageText := 'Command.LanguageCode = {1}',
                        Para1       :=  _command.LanguageCode);
                
END_METHOD

METHOD FB_init : BOOL
VAR_INPUT
  /// if TRUE, the retain variables are initialized (warm start / cold start)
  bInitRetains : BOOL; 
  /// if TRUE, the instance afterwards gets moved into the copy code (online change)
  bInCopyCode  : BOOL;  
END_VAR
                  MyType := 'MC_SwitchLanguageFB';

ExecMode := ExecutionMode.PARALLEL;
Priority := PriorityLevel.NORMAL;
                
END_METHOD

METHOD PROTECTED OnApplyOutCmd
VAR_INPUT
  /// Command message state
  State : CmdMessageState;
END_VAR
                  IF ( State = CmdMessageState.EMPTY ) 
THEN
  // Reset command outputs
  SysDepMemSet(pDest := ADR(OutCmd), Value := 0, DataLen := SIZEOF(OutCmd));         
END_IF

IF (( State = CmdMessageState.ACTIVE ) OR
    ( State = CmdMessageState.DONE   ))
THEN
  // Update results
  OutCmd.ActualLanguageCode := _response.ActualLanguageCode;
END_IF
                
END_METHOD

METHOD PROTECTED OnExecRun : DINT
VAR_IN_OUT
  /// Robot assignment of function
  AxesGroup : AxesGroup; 
END_VAR
                  // call base implementation
SUPER^.OnExecRun(AxesGroup := AxesGroup);

CASE _stepCmd OF
  
  00:  IF ( _execute_R.Q ) AND ( NOT Error)  
       THEN
         // Check function is supported and parameter are valid ?
         IF (( CheckFunctionSupported( AxesGroup := AxesGroup )) AND
             ( CheckParameterValid   ( AxesGroup := AxesGroup )))      
         THEN
           // set busy flag
           Busy := TRUE;
           // Reset command outputs
           SysDepMemSet(pDest := ADR(OutCmd), Value := 0, DataLen := SIZEOF(OutCmd));         
           // apply command parameter
          _parCmd := ParCmd;
           // init parameter sequence
          _command.ParSeq := 1;
           // create command data
           CommandData := CreateCommandPayload(AxesGroup := AxesGroup);
           // Add command to active command register
          _uniqueID := AxesGroup.Acyclic.ActiveCommandRegister.AddCmd( pCommandFB := ADR(THIS^ ));     
           // set timeout
           SetTimeout(PT := _timeoutCmd, rTimer := _timerCmd);
           // inc step counter
          _stepCmd := _stepCmd + 1;
         END_IF 
       END_IF
     

  01:  // Wait for responce received
       IF ( _responseReceived )
       THEN
         // reset response received flag
        _responseReceived := FALSE;
         // update state flags
         OnUpdateStateFlags(_response.State);
         // update state flags
         OnApplyOutCmd(_response.State);

         // Done, Aborted or Error ?
         IF (_response.State >= CmdMessageState.DONE )
         THEN
           // set timeout
           SetTimeout(PT := _timeoutCmd, rTimer := _timerCmd);
           // inc step counter
          _stepCmd := _stepCmd + 1; 
         END_IF
       END_IF


  02: IF ( NOT Execute)
      THEN
        Reset();
      END_IF     

ELSE
  // invalid step
  SetError( ErrorID := RobotLibraryErrorIdEnum.ERR_INVALID_STEP, Overwrite := TRUE );
END_CASE


// Reset FB
IF ( NOT Execute )
THEN
  Reset();
END_IF
                
END_METHOD

METHOD PROTECTED OnUpdateStateFlags
VAR_INPUT
  /// Command message state
  State : CmdMessageState;
END_VAR
                  // Reset State flags
Done := FALSE;

CASE State OF

  // No operation or process is active
  CmdMessageState.EMPTY               :;
  // Created but not yet started
  CmdMessageState.CREATED             :;
  // Buffered and awaiting execution
  CmdMessageState.BUFFERED            : CommandBuffered    := TRUE;
  // Buffered in planner for future execution
  CmdMessageState.BUFFERED_IN_PLANNER : CommandBuffered    := TRUE;
  // Currently active and in progress
  CmdMessageState.ACTIVE              :;                                         
  // Interrupted and awaiting continuation
  CmdMessageState.INTERRUPTED         :;  
  // Requested for abort
  CmdMessageState.ABORT_REQUEST       :;
  // Successfully completed
  CmdMessageState.DONE                : Done               := TRUE;
                                        Busy               := FALSE;
  // Aborted before completion
  CmdMessageState.ABORTED             : Busy               := FALSE;
  // Encountered an error during execution
  CmdMessageState.ERROR               : Error              := TRUE;
                                        Busy               := FALSE;
END_CASE
                
END_METHOD

METHOD INTERNAL ParseResponsePayload : DINT
VAR_INPUT
  /// Response data
  ResponseData : RobotLibraryResponseDataFB;
  /// Timestamp
  Timestamp    : SystemTime;  
END_VAR
VAR
  /// Parameter count
 _parameterCnt : DINT;
END_VAR
// Table 6-77: Received CMD payload (RC to PLC) of "SwitchLanguage"
// --------------------------
// Header
// --------------------------
// Byte 00 : USINT - ParSeq | State     
// Byte 01 : SINT  - AlarmMessageSeverity    
// Byte 02 : UINT  - AlarmMessageCode HB
// Byte 03 :       - AlarmMessageCode LB
// --------------------------
// Datablock
// --------------------------
// Byte 04  : BOOL - SoftMovement
                  // call base implementation to parse the header from payload buffer
ResponseData.PayloadPtr := SUPER^.ParseResponsePayload(ResponseData := ResponseData, Timestamp := Timestamp);

// copy parsed header to response
_response.ParSeq               := _rspHeader.ParSeq;
_response.State                := _rspHeader.State;
_response.AlarmMessageSeverity := _rspHeader.AlarmMessageSeverity;
_response.AlarmMessageCode     := _rspHeader.AlarmMessageCode;


// Check payload remaining ? 
IF ( ResponseData.IsPayloadRemaining)
THEN 
  // Get Response.ActualLanguageCode
 _response.ActualLanguageCode := ResponseData.GetString(2); 
  // inc parameter counter
 _parameterCnt := _parameterCnt + 1;
END_IF


// Create logging
ParseResponsePayloadLog(ResponseData := ResponseData, Timestamp := Timestamp, ParameterCnt := _parameterCnt);
                
END_METHOD

METHOD INTERNAL ParseResponsePayloadLog
VAR_INPUT
  /// Response data
  ResponseData : RobotLibraryResponseDataFB;
  /// Timestamp
  Timestamp    : SystemTime;  
  /// Parameter count
  ParameterCnt : DINT;
END_VAR
                  // Create log entry for Parameter start
CreateLogMessagePara1 ( Timestamp   := Timestamp,
                        MessageType := MessageType.CMD,
                        Severity    := Severity.DEBUG,
                        MessageCode := 0,
                        MessageText := '{1} parameter(s) to parse from the response data:',
                        Para1       := DINT_TO_STRING(ParameterCnt));
                        

// Return if no parameter is remaining...
IF ( ParameterCnt = 0 ) THEN RETURN; END_IF
// dec remaining parameter(s)                        
ParameterCnt := ParameterCnt - 1;
// Create log entry for ActualLanguageCode
CreateLogMessagePara1 ( Timestamp   := Timestamp,
                        MessageType := MessageType.CMD,
                        Severity    := Severity.DEBUG,
                        MessageCode := 0,
                        MessageText := 'Response.ActualLanguageCode = {1}',
                        Para1       := _response.ActualLanguageCode);


                
END_METHOD

METHOD PROTECTED Reset : DINT
VAR_INPUT
END_VAR
                  Reset := SUPER^.Reset();

Done               := FALSE;
Busy               := FALSE;
CommandBuffered    := FALSE;
                
END_METHOD
END_FUNCTION_BLOCK

/// Login on RC from PLC
FUNCTION_BLOCK MC_UserLoginFB EXTENDS RobotLibraryBaseExecuteFB
// ------------------------------------------------------------------------- 
//  SRCI Robot Library                                                
// ------------------------------------------------------------------------- 
//                                                                           
//  Object:      UserLoginFB                                       
//  Author:      Thorsten Brach                                                
//  Date:        2024-06-01
//
//  Description:                                              
//   
//                                                                           
//  Copyright: 
//    (C) 2024 Thorsten Brach. All rights reserved                                                                                                                                            
//             Licensed under the MIT License.
//                                                                           
//  Disclaimer:                                                                           
//    This project is provided without any guarantee and can be used for   
//    private and commercial purposes. Any use is at the user’s 
//    own risk and responsibility.
//
// -------------------------------------------------------------------------
VAR_INPUT
  /// Command parameter 
  ParCmd          : UserLoginParCmd;      
END_VAR
VAR_OUTPUT
  /// Command is transferred and confirmed by the RC
  CommandBuffered : BOOL;
  /// command results
  OutCmd          : UserLoginOutCmd;     
END_VAR

VAR
  /// internal copy of command parameter 
 _parCmd          : UserLoginParCmd;
  /// command data to send
 _command         : UserLoginSendData;
  /// response data received
 _response        : UserLoginRecvData;      
END_VAR

            SUPER^(AxesGroup := AxesGroup);
          

METHOD INTERNAL CheckAddParameter : BOOL
VAR_INPUT
  /// Payload pointer
  PayloadPtr : UDINT;
END_VAR
VAR
  /// Payload as byte array
  Payload    : ARRAY [1..SIZEOF(_command)] OF BYTE;
  /// Null Byte array 
  Null       : ARRAY [1..SIZEOF(_command)] OF BYTE;
  /// Data length to compare
  DataLen    : UDINT;
END_VAR
                  // Payload pointer must be decreased by one byte, because ADR(Payload) is already one byte !
PayloadPtr := LIMIT (0, PayloadPtr - 1, SIZEOF(Payload) -1);
// Convert command struct to payload array
SysDepMemCpy( pDest := ADR(Payload), pSrc := ADR(_command), DataLen := SIZEOF(_command));
// Calculate the data length to compare - at least one byte must be compared !
DataLen := LIMIT(1, SIZEOF(Payload) - PayloadPtr, SIZEOF(Payload)); 
// Compare Payload-Array with Null-Byte-Array
CheckAddParameter := SysDepMemCmp( pData1 := ADR(Payload) + PayloadPtr , pData2 := ADR(Null), DataLen := DataLen) <>  RobotLibraryConstants.OK ;
                
END_METHOD

METHOD PROTECTED CheckFunctionSupported : BOOL
VAR_IN_OUT
  /// Robot assignment of function
  AxesGroup : AxesGroup; 
END_VAR
                  CheckFunctionSupported := AxesGroup.State.RobotData.RCSupportedFunctions.UserLogin;

IF ( NOT CheckFunctionSupported )
THEN
  // call base implementation for set error and create log entry
  SUPER^.CheckFunctionSupported(AxesGroup := AxesGroup);
END_IF
                
END_METHOD

METHOD PROTECTED CheckParameterChanged : BOOL
VAR_IN_OUT
  /// Robot assignment of function
  AxesGroup    : AxesGroup; 
END_VAR
                  // Check ParCmd Size is > 0, because MemCmp does not work correctly with size = 0
IF (SIZEOF(ParCmd) = 0) OR (_stepCmd = 0)
THEN 
  RETURN;
END_IF

// compare memory 
_parameterChanged := ( SysDepMemCmp(pData1 := ADR(ParCmd), pData2 := ADR(_parCmd), DataLen := SIZEOF(ParCmd)) <> RobotLibraryConstants.OK );

// check parameter valid ?
_parameterValid   := CheckParameterValid( AxesGroup := AxesGroup );

IF ((  _parameterChanged        )  AND 
    (  _parameterValid          )) OR
    (  _parameterUpdateInternal )  
THEN  
  // Create log entry for parameter changed event
  CreateLogMessagePara1 ( Timestamp   := AxesGroup.State.SystemTime,
                          MessageType := MessageType.CMD,
                          Severity    := Severity.DEBUG,
                          MessageCode := 0,
                          MessageText := 'NotifyParameterChanged Event {1}',
                          Para1       :=  '' );

  // reset internal flag for send parameter update
 _parameterUpdateInternal := FALSE;
  // update internal copy of parameters 
 _parCmd := ParCmd;
  // inc parameter sequence
 _command.ParSeq := _command.ParSeq + 1;
  // update command data  
  CommandData := CreateCommandPayload(AxesGroup := AxesGroup); // ( Access via reference to rCommandFB in ACR )
  // notify active command register 
  AxesGroup.Acyclic.ActiveCommandRegister.NotifyParameterChanged := _uniqueID;
END_IF
                
END_METHOD

METHOD PROTECTED CheckParameterValid : BOOL
VAR_IN_OUT
  /// Robot assignment of function
  AxesGroup : AxesGroup; 
END_VAR
VAR
  /// internal index for loops
 _idx : DINT;
END_VAR
                  CheckParameterValid := TRUE;


// Check ParCmd.Mode valid ? 
IF (( ParCmd.Mode <> LogonMode.PASSWORD_ONLY         ) AND
    ( ParCmd.Mode <> LogonMode.USERNAME_AND_PASSWORD ) AND
    ( ParCmd.Mode <> LogonMode.LEVEL_ID_AND_PASSWORD ))  
THEN
  // Parameter not valid
  CheckParameterValid := FALSE;
  // Set error
  SetError( ErrorID := RobotLibraryErrorIdEnum.ERR_INVALID_PAR_CMD, Overwrite := TRUE );
  // Create log entry
  CreateLogMessagePara1 ( Timestamp   := AxesGroup.State.SystemTime,
                          MessageType := MessageType.CMD,
                          Severity    := Severity.ERROR,
                          MessageCode := ErrorID,
                          MessageText := 'Invalid Parameter ParCmd.Mode = {1}',
                          Para1       := LOGON_MODE_TO_STRING(ParCmd.Mode));
                       
  RETURN;                          
END_IF

// Check ParCmd.Password valid ? 
IF ( ParCmd.Password = '' )
THEN
  // Parameter not valid
  CheckParameterValid := FALSE;
  // Set error
  SetError( ErrorID := RobotLibraryErrorIdEnum.ERR_INVALID_PAR_CMD, Overwrite := TRUE );
  // Create log entry
  CreateLogMessagePara1 ( Timestamp   := AxesGroup.State.SystemTime,
                          MessageType := MessageType.CMD,
                          Severity    := Severity.ERROR,
                          MessageCode := ErrorID,
                          MessageText := 'Invalid Parameter ParCmd.Password = {1}',
                          Para1       := ParCmd.Password);
                       
  RETURN;                          
END_IF


// Check ParCmd.Username valid ? 
IF ( ParCmd.Username = '' )
THEN
  // Parameter not valid
  CheckParameterValid := FALSE;
  // Set error
  SetError( ErrorID := RobotLibraryErrorIdEnum.ERR_INVALID_PAR_CMD, Overwrite := TRUE );
  // Create log entry
  CreateLogMessagePara1 ( Timestamp   := AxesGroup.State.SystemTime,
                          MessageType := MessageType.CMD,
                          Severity    := Severity.ERROR,
                          MessageCode := ErrorID,
                          MessageText := 'Invalid Parameter ParCmd.Username = {1}',
                          Para1       := ParCmd.Username);
                       
  RETURN;                          
END_IF


